// TwinCAT 3 PLC project Nonplanar_Master
// ProgramVersion: 3.1.4026.20
// libraries:
//   CmpBitmapPool, * (System)
//   Tc2_ControllerToolbox, * (Beckhoff Automation GmbH)
//   Tc2_DataExchange, * (Beckhoff Automation GmbH)
//   Tc2_SerialCom, * (Beckhoff Automation GmbH)
//   Tc2_Standard, * (Beckhoff Automation GmbH)
//   Tc2_System, * (Beckhoff Automation GmbH)
//   Tc2_Utilities, * (Beckhoff Automation GmbH)
//   VisuDialogs, * (System)
//   VisuSymbols,3.5.10.0,System
// project tree:
//   DUTs/ E_NozzleSizeFlow.TcDUT, E_StateExtruder.TcDUT, E_StateSequencer.TcTLEO, ST_ExtruderControl.TcDUT, ST_Hardware_IStepper.TcDUT, ST_HeaterZone.TcDUT, ST_HeaterZone_Parameter.TcDUT, ST_MaterialSettings.TcDUT, ST_MotorControl.TcDUT, ST_PrintingBed.TcDUT, ST_ProgramSequencer.TcDUT, ST_Hardware_QStepper.TcDUT
//   / GlobalTextList.TcGTLO, PlcTask.TcTTO, Visualisierungsmanager.TcVMO (not stored), VISU_TASK.TcTTO
//   GVLs/ GVL_ProgramSequencer.TcGVL, GVL_Instances.TcGVL
//   POUs/Extruder/ FB_ExtruderControl.TcPOU, FB_MotorControl.TcPOU, FB_HeaterZone.TcPOU, FC_ExtrusionCalculations.TcPOU, GVL_Extruder.TcGVL, GVL_HardwareExtruder.TcGVL, GVL_ParameterExtruder.TcGVL, PAR_Extruder.TcGVL
//   POUs/ FB_ProgramSequencer.TcPOU, FC_Instances.TcPOU, MAIN.TcPOU
//   POUs/HexaBridge/ FC_Execute.TcPOU, FC_ExecuteNoWait.TcPOU, FC_WaitForFinish.TcPOU, FC_WriteProgLine.TcPOU, GVL_HexaBridge.TcGVL
//   POUs/PrintingBed/ FB_PrintingBedSync.TcPOU, GVL_PrintingBed.TcGVL
//   VISUs/ ImagePool.TcIPO (not stored), V_Konfiguration.TcVIS, V_Homescreen.TcVIS
// real-time tasks:
//   TASK PlcTask: cycle T#10ms, priority 20, ADS port 350
//   TASK VISU_TASK: cycle T#200000us, priority 30, ADS port 351
// I/O:
//   DEVICE Gerät 1 (EtherCAT) (disabled), AmsNetId 172.16.4.140.2.1
//     Buskoppler Extruder (EK1100) [EK1100 EtherCAT-Koppler (2A E-Bus)]
//       Eingänge (EL1008) [EL1008 8K. Dig. Eingang 24V, 3ms]
//       Ausgänge SSR (EL2004) [EL2004 4K. Dig. Ausgang 24V, 0.5A]
//       Temperatursensoren (EL3204) [EL3204 4Ch. Ana. Input PT100 (RTD)]
//       Stepper Driver STEP (EL2521) [EL2521 1K. Pulse Train Ausgang]
//       Stepper Driver DIR / Enable (EL4132) [EL4132 2Ch. Ana. Ausgang +/-10V, 16bit]
//       Klemme 13 (EL9011) [EL9011 Endklemme]
// variable links:
//   Nonplanar_Master/Nonplanar_Master Instance <-> Device 1 (EtherCAT)/Buskoppler Extruder (EK1100)/Ausgänge SSR (EL2004)
//     PlcTask Outputs/GVL_HardwareExtruder.Q_Activate_Heaters <-> Channel 4/Output
//     PlcTask Outputs/GVL_HardwareExtruder.Q_SSR_Middle <-> Channel 2/Output
//     PlcTask Outputs/GVL_HardwareExtruder.Q_SSR_Nozzle <-> Channel 3/Output
//     PlcTask Outputs/GVL_HardwareExtruder.Q_SSR_Top <-> Channel 1/Output
//   Nonplanar_Master/Nonplanar_Master Instance <-> Device 1 (EtherCAT)/Buskoppler Extruder (EK1100)/Eingänge (EL1008)
//     PlcTask Inputs/GVL_HardwareExtruder.I_PelletsEmpty <-> Channel 1/Input
//   Nonplanar_Master/Nonplanar_Master Instance <-> Device 1 (EtherCAT)/Buskoppler Extruder (EK1100)/Stepper Driver DIR / Enable (EL4132)
//     PlcTask Outputs/GVL_HardwareExtruder.Q_Stepper/nDirection <-> Channel 1/Output
//     PlcTask Outputs/GVL_HardwareExtruder.Q_Stepper/nEnable <-> Channel 2/Output
//   Nonplanar_Master/Nonplanar_Master Instance <-> Device 1 (EtherCAT)/Buskoppler Extruder (EK1100)/Stepper Driver STEP (EL2521)
//     PlcTask Inputs/GVL_HardwareExtruder.I_Stepper/bError <-> PTO Status/Status/Error
//     PlcTask Inputs/GVL_HardwareExtruder.I_Stepper/bStallguardActive <-> PTO Status/Status/Status of input target
//     PlcTask Outputs/GVL_HardwareExtruder.Q_Stepper/nFrequencyValue <-> PTO Control/Frequency value
//   Nonplanar_Master/Nonplanar_Master Instance <-> Device 1 (EtherCAT)/Buskoppler Extruder (EK1100)/Temperatursensoren (EL3204)
//     PlcTask Inputs/GVL_HardwareExtruder.I_TempRaw_Middle <-> RTD Inputs Channel 2/Value
//     PlcTask Inputs/GVL_HardwareExtruder.I_TempRaw_Nozzle <-> RTD Inputs Channel 3/Value
//     PlcTask Inputs/GVL_HardwareExtruder.I_TempRaw_Top <-> RTD Inputs Channel 1/Value

CONFIGURATION Nonplanar_Master
    RESOURCE PLC ON TwinCAT3
        TASK PlcTask(INTERVAL := T#10ms, PRIORITY := 20);
        TASK VISU_TASK(INTERVAL := T#200000us, PRIORITY := 30);
        PROGRAM MAIN WITH PlcTask : MAIN;
        PROGRAM VisuElems_Visu_Prg WITH VISU_TASK : VisuElems.Visu_Prg;
    END_RESOURCE
END_CONFIGURATION

// ---- DUTs/E_NozzleSizeFlow.TcDUT
{attribute 'qualified_only'}
{attribute 'strict'}
// Düsendurchmesser in mm und die zugehärige Reduzierung des maximalen Durchflusses in mm^3/s
TYPE E_NozzleSizeFlow :
(
	fuenf 	:= 0,
	vier	:= -60,
	drei	:= -120,
	zwei 	:= -180,
	ein		:= -240
)DINT := drei;
END_TYPE

// ---- DUTs/E_StateExtruder.TcDUT
{attribute 'qualified_only'}
{attribute 'strict'}
TYPE E_StateExtruder :
(
	OFF			:= 0,
	INIT		:= 10,
	IDLE		:= 100,
	HEATING		:= 200,
	READY		:= 300,
	PRINTING	:= 310,
	SHUTDOWN	:= 400
);
END_TYPE

// ---- DUTs/E_StateSequencer.TcTLEO
{attribute 'qualified_only'}
{attribute 'strict'}
TYPE E_StateSequencer :
(
	OFF					:= 0,
	INIT_1				:= 10,
	INIT_2				:= 11,
	INIT_3				:= 12,
	HOMING_1			:= 90,
	HOMING_2			:= 91,
	
	IDLE				:= 100,
	OPEN_FILE			:= 110,
	CLOSE_FILE			:= 120,
	CHANGE_MATERIAL_1	:= 130,
	CHANGE_MATERIAL_2	:= 131,
	CHANGE_MATERIAL_3	:= 132,
	
	READY				:= 200,
	
	PREP_PRINTING		:= 300,
	PREP_PRINTING_HEX_1	:= 301,
	PREP_PRINTING_HEX_2	:= 302,
	PREP_PRINTING_HEX_3	:= 303,
	PREP_PRINTING_HEX_4 := 304,
	PREP_PRINTING_EXT	:= 305,
	PREP_PRINTING_HEX_5	:= 306,
	PREP_PRINTING_HEX_6	:= 307,
	PREP_PRINTING_HEX_7	:= 308,
	
	READ_FILE			:= 310,
	EXECUTE_LINE		:= 320,
	
	WRITE_KOS			:= 330,
	WRITE_FEED			:= 331,
	WRITE_PROG			:= 335,
	
	EXTRUDER_ON_1		:= 340,
	EXTRUDER_ON_2		:= 341,
	
	EXTRUDER_OFF_1		:= 350,
	START_EXTRUDING		:= 351,
	EXTRUDER_OFF_2		:= 352,
	
	STOP_EXTRUDING		:= 360,
	
	PAUSE				:= 390,
	
	ABORTED				:= 400,
	
	FINISHED			:= 500,
	
	SHUTDOWN			:= 600
);
END_TYPE

// ---- DUTs/ST_ExtruderControl.TcDUT
TYPE ST_ExtruderControl :
STRUCT
	// Steuersignale
	bErrorReset 	: BOOL;						// Reset-Befehl für Fehler
	bStartHeater 	: BOOL;						// Heizelemente aktivieren
	bStopHeater		: BOOL;						// Abschalten und Abkühlen
	bStart 			: BOOL;						// Start-Befehl Extrusion
	bStop 			: BOOL;						// Stop-Befehl Extrusion
	
	// Statusinformationen
	bReady 			: BOOL;						// Betriebsbereit
	bExtruding 		: BOOL;						// Motor läuft
	bHeatingActiv 	: BOOL;						// Heizelemente
	bError 			: BOOL;						// Fehler
	nErrorID      	: UDINT;
    sErrorMsg 		: STRING(80);
END_STRUCT
END_TYPE

// ---- DUTs/ST_Hardware_IStepper.TcDUT
TYPE ST_Hardware_IStepper :
STRUCT
	bStallguardActive 	: BOOL;		// Stallguard nicht aktive --> Motor überlastet
	bError				: BOOL;		// Fehler 
END_STRUCT
END_TYPE

// ---- DUTs/ST_HeaterZone.TcDUT
TYPE ST_HeaterZone :
STRUCT
    // Grunddaten
    bEnabled        : BOOL;                 // Zone aktiv
	fActualTemp   	: LREAL;             	// Isttemperatur [°C]
    fPID_Output     : LREAL;                // PID-Stellgröße [0..100%]
    bAtTemp         : BOOL;                 // Temperatur erreicht
	bErrorReset		: BOOL;					// Fehler zurücksetzen
    bError        	: BOOL;					// Fehler
    nErrorID      	: UDINT;
    sErrorMsg 		: STRING(80);
END_STRUCT
END_TYPE

// ---- DUTs/ST_HeaterZone_Parameter.TcDUT
TYPE ST_HeaterZone_Parameter :
STRUCT
    // PID-Parameter (https://docs.dyzedesign.com/pulsar.html#marlin-firmware)
    fKp             : LREAL 	:= 1.2;       	// Proportionalverstärkung
    fKi             : LREAL  	:= 0.015;   	// Integralverstärkung
    fKd             : LREAL  	:= 50.0;  		// Differentialversträrkung
    fFilterN      	: LREAL 	:= 10.0;		// Filterfaktor für DT1-Anteil des PID-Reglers (zwischen 5 und 20 --> mehr Rauschen = kleiner)
END_STRUCT
END_TYPE

// ---- DUTs/ST_MaterialSettings.TcDUT
TYPE ST_MaterialSettings :
STRUCT
	sMaterial		: STRING(80);		// Materialname	

	fTempPrintingBed: REAL	:= 0;		// <120 [°C]
	
	fTempTop		: LREAL	:= 0;		// <400 [°C]
	fTempMiddle		: LREAL	:= 0;		// <400 [°C]
	fTempNozzle		: LREAL	:= 0;		// <400 [°C]
	
	// https://docs.dyzedesign.com/pulsar.html#flow-to-rpm
	
	fMaxFlowRate	: LREAL := 0;		// Maximaler Volumenstrom [mm^3/s]
	fFlow2RPM		: LREAL := 0;		// Flow to RPM Ratio
	fNozzleSizeCoef	: LREAL := 1;		// Koeffizent Flow2RPM (abhängig von Material und Düse)
END_STRUCT	
END_TYPE

// ---- DUTs/ST_MotorControl.TcDUT
TYPE ST_MotorControl :
STRUCT
	bEnable         	: BOOL		:= FALSE;  	// Freigabe des Motors
	bErrorReset			: BOOL		:= FALSE;	// Fehler zurücksetzen
	bRunning       		: BOOL;					// Motor läuft
	bError        		: BOOL;					// Fehler
    nErrorID      		: UDINT;
    sErrorMsg 			: STRING(80);
END_STRUCT
END_TYPE

// ---- DUTs/ST_PrintingBed.TcDUT
TYPE ST_PrintingBed :
STRUCT
	fSetTemp		: REAL;			// Solltemperatur Druckbett
	fActualTemp		: REAL;			// Isttemperatur Druckbett
	bAtTemp			: BOOL;			// Solltemperatur erreicht (0.5°C Toleranz)
	bErrorReset		: BOOL;
	bError        	: BOOL;			// Fehler
    nErrorID      	: UDINT;
    sErrorMsg 		: STRING(80);
END_STRUCT
END_TYPE

// ---- DUTs/ST_ProgramSequencer.TcDUT
TYPE ST_ProgramSequencer :
STRUCT
	sPath			: STRING(MAX_STRING_LENGTH);// Pfad des Speicherorts des GeoCodes
	
	// Statusinformationen
	bReady 			: BOOL;						// Betriebsbereit
	bPrinting 		: BOOL;						// Druckprozess läuft
	bFinished		: BOOL;						// Druck abgeschlossen
	bError        	: BOOL;						// Fehler
    nErrorID      	: UDINT;
    sErrorMsg 		: STRING(80);
	
	// Steuersignale
	bHeatersEnabled	: BOOL;						// Heizelemente aktiviert --> später Safety Verknüpfung
	bPrintBedClear	: BOOL;						// Druckbett frei?
	bChangeMaterial	: BOOL;						// Extruder starten für Materialwechsel
	bChangeMaterialFinished : BOOL;				// Materialwechsel abschliesen und Extruder anhalten
	bLoadFile		: BOOL;						// File laden
	bCloseFile		: BOOL;						// File schließen
	bStart 			: BOOL;						// Start-Befehl
	bAbort 			: BOOL;						// Drucken abbrechen
	bPause          : BOOL;						// Pausiert Druckprozess
	bResume         : BOOL;						// Druckprozess fortsetzen
	bErrorReset 	: BOOL;						// Reset-Befehl für Fehler
END_STRUCT
END_TYPE

// ---- DUTs/ST_Hardware_QStepper.TcDUT
TYPE ST_Hardware_QStepper :
STRUCT
	nFrequencyValue		: INT;		// Frequenzwert (Bewegunggeschwindigkeit und Richtung) !muss INT sein, nicht UINT!
	nDirection			: INT;		// Legt Bewegungsrichtung fest (16383 entspricht 5V --> gegen den urzeigersinn --> Extrusion, alternativ 0)
	nEnable				: INT;		// Deaktivert Motor wenn aktiv (16383 entspricht 5V --> Motor aus, alternativ 0 entspricht 0V --> Motor an) 
END_STRUCT
END_TYPE

// ---- GVLs/GVL_ProgramSequencer.TcGVL
{attribute 'qualified_only'}
VAR_GLOBAL
	Sequencer		: ST_ProgramSequencer := (sPath := 'C:\Users\Gereon\Desktop\MotionInterface\testpaths\testpath.geo'); 
END_VAR

// ---- GVLs/GVL_Instances.TcGVL
VAR_GLOBAL
	// Befehlsverarbeitung
	Sequencer			: FB_ProgramSequencer;
	
	// Druckbett
	PrintingBed			: FB_PrintingBedSync;

	// Extruder
	ExtruderControl		: FB_ExtruderControl; 
	
	// Heizelemente
	HeaterTop			: FB_HeaterZone;
	HeaterMiddle		: FB_HeaterZone;
	HeaterNozzle		: FB_HeaterZone;
	
	//Motor
	ExtruderMotor		: FB_MotorControl;
END_VAR

// ---- POUs/Extruder/GVL_Extruder.TcGVL
{attribute 'qualified_only'}
VAR_GLOBAL
	Extruder		: ST_ExtruderControl;
	HeaterTop		: ST_HeaterZone;
	HeaterMiddle	: ST_HeaterZone;	
	HeaterNozzle	: ST_HeaterZone;
	ExtruderMotor	: ST_MotorControl;
END_VAR

// ---- POUs/Extruder/GVL_HardwareExtruder.TcGVL
{attribute 'qualified_only'}
VAR_GLOBAL
	// EL3204 – RTD-Temperatureingänge (Heizelemente)
	I_TempRaw_Top  		AT %I* : INT;  
	I_TempRaw_Middle 	AT %I* : INT;   
	I_TempRaw_Nozzle  	AT %I* : INT;    

	// EL2004 – Digitale Ausgänge (Heizelemente)
	Q_SSR_Top      		AT %Q* : BOOL;   
	Q_SSR_Middle    	AT %Q* : BOOL;   
	Q_SSR_Nozzle    	AT %Q* : BOOL;  
	Q_Activate_Heaters	AT %Q* : BOOL;

	// EL2521 – Pulsausgabe (Stepper Motor Driver)
	Q_Stepper	  		AT %Q* : ST_Hardware_QStepper;		
	I_Stepper  			AT %I* : ST_Hardware_IStepper;
	
	// EL1002 – Digitale Eingänge
	I_PelletsEmpty      AT %I* : BOOL;    	//Materialzuführung leer
END_VAR

// ---- POUs/Extruder/GVL_ParameterExtruder.TcGVL
{attribute 'qualified_only'}
VAR_GLOBAL PERSISTENT // Speichern der Online-Veränderungen
	// Mehr Informationen unter: https://docs.dyzedesign.com/pulsar.html#slicer-and-print-settings	

	// Materialabhängige Eigenschaften
	{attribute 'TcInitOnReset'} // Neuladen bei Kalt Reset (oben rechts)
	aMaterialSettings	: ARRAY[1..20] OF ST_MaterialSettings := [
			(sMaterial := 'Test-Material', 	fTempPrintingBed := 30, fTempTop := 201, 	fTempMiddle := 201, fTempNozzle := 201,	fMaxFlowRate := 600, fFlow2RPM := 0.65, fNozzleSizeCoef := 1.10),
			(sMaterial := 'PETG', 			fTempPrintingBed := 90, fTempTop := 101, 	fTempMiddle := 241, fTempNozzle := 231, fMaxFlowRate := 592, fFlow2RPM := 0.75,	fNozzleSizeCoef := 1.10),
			(sMaterial := 'PLA', 			fTempPrintingBed := 60, fTempTop := 101, 	fTempMiddle := 221, fTempNozzle := 211, fMaxFlowRate := 607, fFlow2RPM := 0.55,	fNozzleSizeCoef := 1.35),
			(sMaterial := 'PC-ABS-CF', 		fTempPrintingBed := 110,fTempTop := 301, 	fTempMiddle := 301, fTempNozzle := 301, fMaxFlowRate := 700, fFlow2RPM := 0.58, fNozzleSizeCoef := 1.10),
			(sMaterial := 'ABS', 			fTempPrintingBed := 90,	fTempTop := 131	, 	fTempMiddle := 231, fTempNozzle := 231, fMaxFlowRate := 658, fFlow2RPM := 0.65, fNozzleSizeCoef := 1.05), 
			15(())]; // Speichert materialabhängige Extrudereinstellungen (neues Material: Zeile oben kopieren, einfügen und Zähler reduzieren)		
	{attribute 'TcInitOnReset'} // Neuladen bei Kalt Reset (oben rechts)
	nMaterial		: UINT				:= 5;			// Aktuell gewähltes Material
		
	nNozzleSize		: E_NozzleSizeFlow	:= E_NozzleSizeFlow.vier; // Düsendurchmesser [mm] als Wort entspricht der Reduzierung des Durchflusses [mm^3/s]
	fLayerWidth     : LREAL 			:= 5.0;			// Schichtbreite [mm]
	fLayerHeight    : LREAL 			:= 1.0;			// Schichthöhe [mm]
	fSpeedOverride  : LREAL 			:= 10.0; 		// [%] Geschwindigkeits-Override in Prozent der Maximalgeschwindigkeit
	fSafetyMargin	: LREAL				:= 75.0;		// [%] Sicherheitsfaktor für die maximale Druckgeschwindigkeit (75%)
	
	// Berechnete Werte - siehe FC_ExtrusionCalculation
	fMaximumFlow	: LREAL				:= 0;			// Maximaler Durchfluss mit Abzug der Beschränkungen durch die Düse [mm^3/s]
	fMaximumSpeed	: LREAL				:= 0;			// Maximale Druckgeschwindigkeit [mm/s]
	fFlowRate		: LREAL				:= 0;			// Durchfluss [mm^3/s]
	fMotorRPM		: LREAL				:= 0;			// Notwendige RPM des Motors
	
	// Verfahrgeschwindigkeit
	fTravelSpeed	: LREAL				:= 100;			// Verfahrgeschwindigkeit [mm/s]
	
	// PID-Regler Heizelemente
	WarmupHeaterTop		: ST_HeaterZone_Parameter;
	WarmupHeaterMiddle	: ST_HeaterZone_Parameter;	
	WarmupHeaterNozzle	: ST_HeaterZone_Parameter;
	PrintingHeaterTop	: ST_HeaterZone_Parameter;
	PrintingHeaterMiddle: ST_HeaterZone_Parameter;	
	PrintingHeaterNozzle: ST_HeaterZone_Parameter;
	
	tRampTime		: TIME				:= T#3M;		// Länge der Rampe bei Sprüngen
	nPIDCycleFactor	: UINT  			:= 10;			// PID rechnet alle n Zyklen
    tPWM_Period     : TIME  			:= T#3S;        // PWM-Periode SSR
    fAtTempTolerance: LREAL 			:= 50.0;         // Toleranz für Signal Temperatur erreicht [°C]
END_VAR

// ---- POUs/Extruder/PAR_Extruder.TcGVL
{attribute 'qualified_only'}
VAR_GLOBAL CONSTANT
	// Nicht bearbeiten!
	// Quelle: https://docs.dyzedesign.com/pulsar.html#marlin-firmware	

	// Temperatur
    C_MAX_SET_TEMP		: LREAL := 400.0;		// Maximale Setzbare Temperaturgrenze [°C]
    C_MIN_SET_TEMP		: LREAL := 0;			// Minimal Setzbare Temperaturgrenze [°C]
	C_MAX_SENSOR_TEMP	: LREAL := 505.0;		// Maximale Plausibilitätsgrenze Sensoren [°C]
    C_MIN_SENSOR_TEMP	: LREAL := 0;			// Minimale Plausibilitätsgrenze Sensoren [°C]
	C_MAX_TEMP			: LREAL := 500.0;		// Maximaltemperatur Extruder [°C]
	
	// Stepper Driver 
	C_MAX_RPM_SCREW		: LREAL := 60;			// Maximale zulässige RPM --> Anpassung: EL2521 Grundfrequenz
	C_MAX_RPM_SCREW_FULL: LREAL := 50;			// Maximale zulässige RPM mit Material
	C_GEAR_RATIO		: LREAL := 11.46;		// Übersetzung Motor --> Schraube
	C_STEPPER_DIR		: BOOL	:= FALSE;		// Drehrichtung
END_VAR

// ---- POUs/HexaBridge/GVL_HexaBridge.TcGVL
{attribute 'qualified_only' := 'FALSE'}
//  GVL_HexaBridge  -  Globale Variablen für ADS-HexaBOF-Bridge
VAR_GLOBAL
    // Befehlsschnittstelle
    sCommand        : STRING(255);          // Befehlsname
    sParameter      : STRING(1000);         // Parameter-String
    bExecute        : BOOL;                 // Steigende Flanke = Befehl ausführen
	bCommandSent	: BOOL;					// Befehl gesendet
    bBusy           : BOOL;                 // Bridge verarbeitet Befehl
    bDone           : BOOL;                 // Befehl abgeschlossen
    bError          : BOOL;                 // Fehler aufgetreten
    nErrorCode      : INT;                  // Fehlercode (0=OK)
    sErrorMsg       : STRING(255);          // Fehlermeldung
    sResult         : STRING(1000);         // Ergebnis-String

    // Status
    bHexConnected   : BOOL;                 // HexaBOF verbunden
    bBridgeRunning  : BOOL;                 // Python-Bridge aktiv

    // Direkte GEO-Strings
    sGeoLine        : STRING(1000);         // Einzel-GEO-Zeile
    sGeoBlock       : STRING(10000);        // GEO-Block (mehrzeilig)
	
	// Programm Block schreiben im Hintergrund, um diesen später auszuführen
	sProgLine		: STRING(1000);         // Einzel-GEO-Zeile zu Programm hinzufügen
	bProgLineReady	: BOOL;        			// Zeile bereit zum schreiben
	bProgLineSaved	: BOOL;        			// Zeile gespeichert
	bProgLineExecution : BOOL;        		// Blockiert das Schreiben neuer Programmzeilen beim Starten des Ausführens eines Blocks
END_VAR

// ---- POUs/PrintingBed/GVL_PrintingBed.TcGVL
{attribute 'qualified_only'}
VAR_GLOBAL
	PrintingBed		: ST_PrintingBed;
END_VAR

// ---- POUs/MAIN.TcPOU
PROGRAM MAIN
VAR
END_VAR

FC_Instances();

END_PROGRAM

// ---- POUs/FC_Instances.TcPOU
FUNCTION FC_Instances : BOOL
VAR_INPUT
END_VAR
VAR
END_VAR

// Befehlsverarbeitung
Sequencer(
	sPath			:= GVL_ProgramSequencer.Sequencer.sPath,
	bPelletsEmpty	:= GVL_HardwareExtruder.I_PelletsEmpty,
	bReady 			=> GVL_ProgramSequencer.Sequencer.bReady,
	bPrinting 		=> GVL_ProgramSequencer.Sequencer.bPrinting,
	bFinished		=> GVL_ProgramSequencer.Sequencer.bFinished,
	bError        	=> GVL_ProgramSequencer.Sequencer.bError,
	nErrorID      	=> GVL_ProgramSequencer.Sequencer.nErrorID,
	sErrorMsg 		=> GVL_ProgramSequencer.Sequencer.sErrorMsg,
	bHeatersEnabled	:= GVL_ProgramSequencer.Sequencer.bHeatersEnabled,
	bPrintBedClear	:= GVL_ProgramSequencer.Sequencer.bPrintBedClear,
	bChangeMaterial	:= GVL_ProgramSequencer.Sequencer.bChangeMaterial,
	bChangeMaterialFinished := GVL_ProgramSequencer.Sequencer.bChangeMaterialFinished,
	bLoadFile		:= GVL_ProgramSequencer.Sequencer.bLoadFile,
	bCloseFile		:= GVL_ProgramSequencer.Sequencer.bCloseFile,
	bStart 			:= GVL_ProgramSequencer.Sequencer.bStart,
	bAbort 			:= GVL_ProgramSequencer.Sequencer.bAbort,
	bPause          := GVL_ProgramSequencer.Sequencer.bPause,
	bResume         := GVL_ProgramSequencer.Sequencer.bResume,
	bErrorReset 	:= GVL_ProgramSequencer.Sequencer.bErrorReset);

// Druckbett
PrintingBed(
	bErrorReset		:= GVL_PrintingBed.PrintingBed.bErrorReset,
	bError			=> GVL_PrintingBed.PrintingBed.bError,
	nErrorID		=> GVL_PrintingBed.PrintingBed.nErrorID,
	sErrorMsg		=> GVL_PrintingBed.PrintingBed.sErrorMsg);

// Extruder	
ExtruderControl(
	bErrorReset		:= GVL_Extruder.Extruder.bErrorReset,
	bHeatersEnabled := GVL_ProgramSequencer.Sequencer.bHeatersEnabled,
	bReady			=> GVL_Extruder.Extruder.bReady,
	bExtruding		=> GVL_Extruder.Extruder.bExtruding,
	bHeatingActiv	=> GVL_Extruder.Extruder.bHeatingActiv,
	bError			=> GVL_Extruder.Extruder.bError,
	nErrorID      	=> GVL_Extruder.Extruder.nErrorID,
    sErrorMsg 		=> GVL_Extruder.Extruder.sErrorMsg,
	bStartHeater	:= GVL_Extruder.Extruder.bStartHeater,
	bStopHeater		:= GVL_Extruder.Extruder.bStopHeater,
	bStart			:= GVL_Extruder.Extruder.bStart,
	bStop			:= GVL_Extruder.Extruder.bStop);	

// Heizelemente
HeaterTop(
	bEnable			:= GVL_Extruder.HeaterTop.bEnabled,
    fSetTemp		:= GVL_ParameterExtruder.aMaterialSettings[GVL_ParameterExtruder.nMaterial].fTempTop,
	fPID_Output     => GVL_Extruder.HeaterTop.fPID_Output,
	bAtTemp         => GVL_Extruder.HeaterTop.bAtTemp,
    bErrorReset		:= GVL_Extruder.HeaterTop.bErrorReset,
    bError        	=> GVL_Extruder.HeaterTop.bError,
    nErrorID      	=> GVL_Extruder.HeaterTop.nErrorID,
    sErrorMsg 		=> GVL_Extruder.HeaterTop.sErrorMsg,
	fWarmupKp       := GVL_ParameterExtruder.WarmupHeaterTop.fKp,
	fWarmupKi       := GVL_ParameterExtruder.WarmupHeaterTop.fKi,
	fWarmupKd       := GVL_ParameterExtruder.WarmupHeaterTop.fKd,
	fWarmupFilterN 	:= GVL_ParameterExtruder.WarmupHeaterTop.fFilterN,
	bPrinting		:= GVL_Extruder.Extruder.bExtruding,
	fPrintingKp     := GVL_ParameterExtruder.PrintingHeaterTop.fKp,
	fPrintingKi     := GVL_ParameterExtruder.PrintingHeaterTop.fKi,
	fPrintingKd     := GVL_ParameterExtruder.PrintingHeaterTop.fKd,
	fPrintingFilterN:= GVL_ParameterExtruder.PrintingHeaterTop.fFilterN,
	tRampTime		:= GVL_ParameterExtruder.tRampTime,
	nPIDCycleFactor	:= GVL_ParameterExtruder.nPIDCycleFactor,
	tPWM_Period     := GVL_ParameterExtruder.tPWM_Period,
	fAtTempTolerance:= GVL_ParameterExtruder.fAtTempTolerance,
	nTempRaw		:= GVL_HardwareExtruder.I_TempRaw_Top,
	fActualTemp		=> GVL_Extruder.HeaterTop.fActualTemp,
	bSSR_Out		=> GVL_HardwareExtruder.Q_SSR_Top);

HeaterMiddle(
	bEnable			:= GVL_Extruder.HeaterMiddle.bEnabled,
    fSetTemp		:= GVL_ParameterExtruder.aMaterialSettings[GVL_ParameterExtruder.nMaterial].fTempMiddle,
	fPID_Output     => GVL_Extruder.HeaterMiddle.fPID_Output,
	bAtTemp         => GVL_Extruder.HeaterMiddle.bAtTemp,
    bErrorReset		:= GVL_Extruder.HeaterMiddle.bErrorReset,
    bError        	=> GVL_Extruder.HeaterMiddle.bError,
    nErrorID      	=> GVL_Extruder.HeaterMiddle.nErrorID,
    sErrorMsg 		=> GVL_Extruder.HeaterMiddle.sErrorMsg,
	fWarmupKp       := GVL_ParameterExtruder.WarmupHeaterMiddle.fKp,
	fWarmupKi       := GVL_ParameterExtruder.WarmupHeaterMiddle.fKi,
	fWarmupKd       := GVL_ParameterExtruder.WarmupHeaterMiddle.fKd,
	fWarmupFilterN 	:= GVL_ParameterExtruder.WarmupHeaterMiddle.fFilterN,
	bPrinting		:= GVL_Extruder.Extruder.bExtruding,
	fPrintingKp     := GVL_ParameterExtruder.PrintingHeaterMiddle.fKp,
	fPrintingKi     := GVL_ParameterExtruder.PrintingHeaterMiddle.fKi,
	fPrintingKd     := GVL_ParameterExtruder.PrintingHeaterMiddle.fKd,
	fPrintingFilterN:= GVL_ParameterExtruder.PrintingHeaterMiddle.fFilterN,
	tRampTime		:= GVL_ParameterExtruder.tRampTime,
	nPIDCycleFactor	:= GVL_ParameterExtruder.nPIDCycleFactor,  
	tPWM_Period     := GVL_ParameterExtruder.tPWM_Period,      
	fAtTempTolerance:= GVL_ParameterExtruder.fAtTempTolerance,
	nTempRaw		:= GVL_HardwareExtruder.I_TempRaw_Middle,
	fActualTemp		=> GVL_Extruder.HeaterMiddle.fActualTemp,
	bSSR_Out		=> GVL_HardwareExtruder.Q_SSR_Middle);
		
HeaterNozzle(
	bEnable			:= GVL_Extruder.HeaterNozzle.bEnabled,
    fSetTemp		:= GVL_ParameterExtruder.aMaterialSettings[GVL_ParameterExtruder.nMaterial].fTempNozzle,
	fPID_Output     => GVL_Extruder.HeaterNozzle.fPID_Output,
	bAtTemp         => GVL_Extruder.HeaterNozzle.bAtTemp,
    bErrorReset		:= GVL_Extruder.HeaterNozzle.bErrorReset,
    bError        	=> GVL_Extruder.HeaterNozzle.bError,
    nErrorID      	=> GVL_Extruder.HeaterNozzle.nErrorID,
    sErrorMsg 		=> GVL_Extruder.HeaterNozzle.sErrorMsg,
	fWarmupKp       := GVL_ParameterExtruder.WarmupHeaterNozzle.fKp,
	fWarmupKi       := GVL_ParameterExtruder.WarmupHeaterNozzle.fKi,
	fWarmupKd       := GVL_ParameterExtruder.WarmupHeaterNozzle.fKd,
	fWarmupFilterN 	:= GVL_ParameterExtruder.WarmupHeaterNozzle.fFilterN,
	bPrinting		:= GVL_Extruder.Extruder.bExtruding,
	fPrintingKp     := GVL_ParameterExtruder.PrintingHeaterNozzle.fKp,
	fPrintingKi     := GVL_ParameterExtruder.PrintingHeaterNozzle.fKi,
	fPrintingKd     := GVL_ParameterExtruder.PrintingHeaterNozzle.fKd,
	fPrintingFilterN:= GVL_ParameterExtruder.PrintingHeaterNozzle.fFilterN,
	tRampTime		:= GVL_ParameterExtruder.tRampTime,
	nPIDCycleFactor	:= GVL_ParameterExtruder.nPIDCycleFactor,  
	tPWM_Period     := GVL_ParameterExtruder.tPWM_Period,      
	fAtTempTolerance:= GVL_ParameterExtruder.fAtTempTolerance,
	nTempRaw		:= GVL_HardwareExtruder.I_TempRaw_Nozzle,
	fActualTemp		=> GVL_Extruder.HeaterNozzle.fActualTemp,
	bSSR_Out		=> GVL_HardwareExtruder.Q_SSR_Nozzle);

//Motor
ExtruderMotor(
	bEnable			:= GVL_Extruder.ExtruderMotor.bEnable,
	bErrorReset		:= GVL_Extruder.ExtruderMotor.bErrorReset,
	fSetRPM			:= GVL_ParameterExtruder.fMotorRPM,
	bError_Stepper	:= GVL_HardwareExtruder.I_Stepper.bError,
	bStepper_STALL	:= GVL_HardwareExtruder.I_Stepper.bStallguardActive,
	bRunning		=> GVL_Extruder.ExtruderMotor.bRunning,
	bError			=> GVL_Extruder.ExtruderMotor.bError,
	nErrorID		=> GVL_Extruder.ExtruderMotor.nErrorID,
	sErrorMsg		=> GVL_Extruder.ExtruderMotor.sErrorMsg,
	nPTO_FreqValue	=> GVL_HardwareExtruder.Q_Stepper.nFrequencyValue,
	n_Direction		=> GVL_HardwareExtruder.Q_Stepper.nDirection,
	n_Enable		=> GVL_HardwareExtruder.Q_Stepper.nEnable);

END_FUNCTION

// ---- POUs/FB_ProgramSequencer.TcPOU
FUNCTION_BLOCK FB_ProgramSequencer
VAR_INPUT
	sPath			: STRING(MAX_STRING_LENGTH);// Pfad des Speicherorts des GeoCodes
	bPelletsEmpty	: BOOL;						// Feeding System meldet, dass keine Pellets am Extruder ankommen
END_VAR
VAR_OUTPUT
	// Statusinformationen
	bReady 			: BOOL;						// Betriebsbereit
	bPrinting 		: BOOL;						// Druckprozess läuft
	bFinished		: BOOL;						// Druck abgeschlossen
	bError        	: BOOL;						// Fehler
    nErrorID      	: UDINT;
    sErrorMsg 		: STRING(80);
END_VAR
VAR
	// Zustandsmaschine
	eState			: E_StateSequencer := E_StateSequencer.OFF;	// Zustand
	eLastState		: E_StateSequencer := E_StateSequencer.OFF; // Vorheriger zustand
	bFirstRunState	: BOOL;						// Erster Durchlauf des Zusands nach einem Zusandswechsel
	
	// Dateiverarbeitung
	fbOpenFile		: FB_FileOpen;
	fbReadFile		: FB_FileGets;
	fbCloseFile		: FB_FileClose;
	hFile  			: UINT;						// file handle
	bFileLoaded		: BOOL;						// Datei geladen
	sLine 			: STRING(MAX_STRING_LENGTH);// Speicher für die gelesene Zeile
	sLineTrimmed	: STRING(MAX_STRING_LENGTH);
	
	// Programmablauf
	bProgBlockStart			: BOOL;				// Erster Befehl des Programmblocks
	bBlockWithExt			: BOOL;				// Extruder in Programmblock aktiv
	bStopExtOnBlockEnd 		: BOOL;				// Extruder am Blockende ausschalten
	bBackToExtruderOn2	 	: BOOL;				// Rücksprung nach Anhalten des Extruders
	bBackToPause			: BOOL;				// Rücksprung nach Anhalten des Extruders
	
	// Änderung Vorschubgeschwindigkeit
	fFeed			: LREAL;
	fTravelFeed		: LREAL;
	bDryRun: BOOL := TRUE;
END_VAR
VAR_IN_OUT
	// Steuersignale
	bHeatersEnabled	: BOOL;						// Heizelemente aktiviert
	bPrintBedClear	: BOOL;						// Druckbett frei?
	bChangeMaterial	: BOOL;						// Extruder starten für Materialwechsel
	bChangeMaterialFinished : BOOL;				// Materialwechsel abschliesen und Extruder anhalten
	bLoadFile		: BOOL;						// File laden
	bCloseFile		: BOOL;						// File schließen
	bStart 			: BOOL;						// Start-Befehl
	bAbort 			: BOOL;						// Drucken abbrechen
	bPause          : BOOL;						// Pausiert Druckprozess
	bResume         : BOOL;						// Druckprozess fortsetzen
	bErrorReset 	: BOOL;						// Reset-Befehl für Fehler
END_VAR

// Schritte: DUTs/E_StateSequencer

// =============================================================================
// Zustandsmaschine
// =============================================================================
IF eLastState <> eState THEN
	bFirstRunState := TRUE;
ELSE
	bFirstRunState := FALSE;
END_IF
eLastState := eState;

// =============================================================================
// Funktionsabhängigkeiten
// =============================================================================
IF bPelletsEmpty THEN
	bPause := TRUE;
	sErrorMsg := 'Feeding System meldet, dass keine Pellets am Extruder ankommen';
END_IF

IF bAbort OR bPause THEN
	bStart := FALSE;
END_IF

IF NOT bHeatersEnabled THEN
	GVL_Extruder.Extruder.bStopHeater := TRUE;
END_IF

IF bResume THEN
	bPause := FALSE;
END_IF

GVL_HardwareExtruder.Q_Activate_Heaters := bHeatersEnabled;

// =============================================================================
// Fehlerbahandlung
// =============================================================================

// Da absolut nichts angeschlossen ist, zwingen wir im Trockenlauf ALLE 
// Hardware-Komponenten auf "fehlerfrei" und "betriebsbereit"!
IF bDryRun THEN
	
	// A. HexaBridge Spoofing
	GVL_HexaBridge.bError := FALSE;
	GVL_HexaBridge.nErrorCode := 0;
	GVL_HexaBridge.sErrorMsg := '';
	GVL_HexaBridge.bHexConnected := TRUE;
	GVL_HexaBridge.bBridgeRunning := TRUE;
	
	// B. Extruder Spoofing (Fehlerfrei & sofort heiß)
	GVL_Extruder.Extruder.bError := FALSE;
	GVL_Extruder.Extruder.nErrorID := 0;
	GVL_Extruder.Extruder.sErrorMsg := '';
	GVL_Extruder.Extruder.bReady := TRUE;
	// Wenn TwinCAT heizen will, tun wir so, als wäre er sofort heiß:
	IF bHeatersEnabled THEN 
		GVL_Extruder.Extruder.bHeatingActiv := TRUE; 
	END_IF

	// C. Druckbett Spoofing (Fehlerfrei & Zieltemperatur erreicht)
	GVL_PrintingBed.PrintingBed.bError := FALSE;
	GVL_PrintingBed.PrintingBed.nErrorID := 0;
	GVL_PrintingBed.PrintingBed.sErrorMsg := '';
	// Wenn eine Zieltemperatur > 0 gesetzt wird, geben wir sofort das "Ist warm!" Signal:
	IF GVL_PrintingBed.PrintingBed.fSetTemp > 0.0 THEN
		GVL_PrintingBed.PrintingBed.bAtTemp := TRUE;
	ELSE
		GVL_PrintingBed.PrintingBed.bAtTemp := FALSE;
	END_IF

END_IF


// Fehler zurücksetzen
IF bErrorReset AND bError THEN
	GVL_Extruder.Extruder.bErrorReset := TRUE;
	GVL_PrintingBed.PrintingBed.bErrorReset := TRUE;
	
	// HexaBridge reset
	GVL_HexaBridge.bExecute := FALSE;
	GVL_HexaBridge.bError := FALSE;
	GVL_HexaBridge.nErrorCode := 0;
	GVL_HexaBridge.sErrorMsg := '';
	
	bErrorReset := FALSE;
	bError := FALSE;
	nErrorID := 0;
	sErrorMsg := '';
ELSIF bErrorReset AND NOT bError THEN
	sErrorMsg := '';
END_IF

// Fehler zusammenführen
bError := bError 
	OR GVL_Extruder.Extruder.bError
	OR GVL_HexaBridge.bError
	OR GVL_PrintingBed.PrintingBed.bError;

// Fehlernachrichten zusammenführen
IF bError THEN
	IF GVL_Extruder.Extruder.bError			THEN nErrorID := GVL_Extruder.Extruder.nErrorID; END_IF
	IF GVL_HexaBridge.bError				THEN nErrorID := TO_UDINT(GVL_Hexabridge.nErrorCode); END_IF
	IF GVL_PrintingBed.PrintingBed.bError	THEN nErrorID := GVL_PrintingBed.PrintingBed.nErrorID; END_IF
	
	IF GVL_Extruder.Extruder.bError			THEN sErrorMsg := GVL_Extruder.Extruder.sErrorMsg; END_IF
	IF GVL_HexaBridge.bError				THEN sErrorMsg := GVL_Hexabridge.sErrorMsg; END_IF
	IF GVL_PrintingBed.PrintingBed.bError	THEN sErrorMsg := GVL_PrintingBed.PrintingBed.sErrorMsg; END_IF
END_IF

// Zusandswechsel im Fehlerfall
IF bError AND NOT (eState = E_StateSequencer.IDLE 
				OR eState = E_StateSequencer.OFF 
				OR eState = E_StateSequencer.READY
				OR eState = E_StateSequencer.SHUTDOWN) THEN
	IF eState < E_StateSequencer.IDLE THEN
		eState := E_StateSequencer.OFF;
	ELSIF eState > E_StateSequencer.READY AND eState < E_StateSequencer.ABORTED THEN
		GVL_Extruder.Extruder.bStopHeater := TRUE;
		bHeatersEnabled := FALSE;
		bAbort := TRUE;
		eState := E_StateSequencer.ABORTED;
	END_IF
END_IF

IF (NOT GVL_Hexabridge.bBridgeRunning OR NOT GVL_Hexabridge.bHexConnected)
AND eState >= E_StateSequencer.READY THEN
	eState := E_StateSequencer.OFF;
	bError := TRUE;
	sErrorMsg := 'HexaBridge ist nicht verbunden!';
END_IF

// =============================================================================
// Status
// =============================================================================
bPrinting := GVL_Extruder.Extruder.bExtruding OR GVL_Extruder.Extruder.bReady;

// =============================================================================
// Vorschubgeschwindigkeit
// =============================================================================
fFeed := GVL_ParameterExtruder.fMaximumSpeed;
fTravelFeed := GVL_ParameterExtruder.fTravelSpeed;

// =============================================================================
// Zustandsmaschine
// =============================================================================
CASE eState OF
	// =============================================================================
	E_StateSequencer.OFF : // Ausgeschaltet
	// =============================================================================
		// Alles aus
		GVL_Extruder.Extruder.bStartHeater := FALSE;
		GVL_Extruder.Extruder.bStopHeater := TRUE;
		GVL_Extruder.Extruder.bStart := FALSE;
		GVL_Extruder.Extruder.bStop := TRUE;
		GVL_PrintingBed.PrintingBed.fSetTemp := 0.0;
	
		// Status
		bReady := FALSE;
		
		IF NOT bError THEN
			eState := E_StateSequencer.INIT_1;
		END_IF
	
	// =============================================================================
	E_StateSequencer.INIT_1: // Initialisierung
	// =============================================================================
		IF GVL_HexaBridge.bHexConnected AND GVL_HexaBridge.bBridgeRunning THEN
			eState := E_StateSequencer.INIT_2;
		END_IF
		
	// =============================================================================
	E_StateSequencer.INIT_2: // Koordinatensystem setzen
	// =============================================================================
		IF FC_Execute('GEO_LINE','SK Extruder') THEN
			eState := E_StateSequencer.INIT_3;
		END_IF
		
	// =============================================================================
	E_StateSequencer.INIT_3: // Kardanwinkel auswählen
	// =============================================================================
		IF FC_Execute('GEO_LINE','NF 2') THEN
			eState := E_StateSequencer.HOMING_1;
		END_IF
	
	// =============================================================================
	E_StateSequencer.HOMING_1: // Verfahrgeschwindigkeit setzen
	// =============================================================================
		IF FC_Execute('GEO_LINE',CONCAT('VF ',TO_STRING(fTravelFeed * 60))) THEN // Vorschub [mm/min]
			eState := E_StateSequencer.HOMING_2;
		END_IF
	
	// =============================================================================
	E_StateSequencer.HOMING_2: // Home Position anfahren (Einfahren)
	// =============================================================================
		IF FC_Execute('GEO_LINE','PU') THEN
			eState := E_StateSequencer.IDLE;
		END_IF
	
	// =============================================================================
	E_StateSequencer.IDLE : // Idle (Keine Datei geöffnet)
	// =============================================================================
		// Alles aus
		GVL_Extruder.Extruder.bStartHeater := FALSE;
		GVL_Extruder.Extruder.bStart := FALSE;
	
		// Status
		bReady := FALSE;
		
		IF bChangeMaterial THEN
			eState := E_StateSequencer.CHANGE_MATERIAL_1;
		ELSIF bFileLoaded THEN 
			eState := E_StateSequencer.READY;
		ELSIF bLoadFile THEN
			eState := E_StateSequencer.OPEN_FILE;
		END_IF
	
	// =============================================================================
	E_StateSequencer.OPEN_FILE : // File öffnen
	// =============================================================================
		IF bFirstRunState THEN
			fbOpenFile(
				sNetId := '', 
				sPathName := sPath, 
				nMode := FOPEN_MODEREAD, 
				bExecute := TRUE, 
				tTimeout := T#5S);
		ELSE
			fbOpenFile(bExecute := FALSE);
		END_IF
			
		IF fbOpenFile.bError THEN
			bError := TRUE;
			nErrorID := 3001;
			sErrorMsg := 'Datei: Fehler beim oeffnen der Datei';
		END_IF
		
		IF NOT bFirstRunState AND NOT fbOpenFile.bBusy AND NOT fbOpenFile.bError AND fbOpenFile.hFile <> 0 THEN
			hFile := fbOpenFile.hFile;
			bFileLoaded := TRUE;
			bLoadFile := FALSE;
			eState := E_StateSequencer.READY;
		END_IF

	// =============================================================================
	E_StateSequencer.CLOSE_FILE : // File schließen
	// =============================================================================
		IF bFirstRunState AND hFile <> 0 THEN
			fbCloseFile(
				sNetId := '',
  				hFile := hFile,
				bExecute := TRUE, 
				tTimeout := T#5S);
		ELSE
			fbCloseFile(bExecute := FALSE);
		END_IF
		
		IF fbCloseFile.bError THEN
			bError := TRUE;
			nErrorID := 3002;
			sErrorMsg := 'Datei: Fehler beim schliessen der Datei';
		END_IF
		
		IF (NOT bFirstRunState AND NOT fbCloseFile.bBusy AND NOT fbCloseFile.bError) 
		OR hFile = 0 THEN
			hFile := 0;
			bFileLoaded := FALSE;
			bCloseFile := FALSE;
			eState := E_StateSequencer.IDLE;
		END_IF
		
	// =============================================================================
	E_StateSequencer.CHANGE_MATERIAL_1 : // Extruder aufheizen
	// =============================================================================
		bChangeMaterial := FALSE;
	
		// Heizungen aktivieren
		IF bHeatersEnabled THEN
			GVL_Extruder.Extruder.bStopHeater := FALSE;
			GVL_Extruder.Extruder.bStartHeater := TRUE;
		END_IF
		
		//Status
		bPrintBedClear := FALSE;
		
		IF bAbort THEN
			eState := E_StateSequencer.ABORTED;		
		ELSIF GVL_Extruder.Extruder.bReady THEN
			eState := E_StateSequencer.CHANGE_MATERIAL_2;
		END_IF
		
	// =============================================================================
	E_StateSequencer.CHANGE_MATERIAL_2 : // Extrudieren bis zum Beenden
	// =============================================================================
		// Extruder aktivieren
		GVL_Extruder.Extruder.bStop := FALSE;
		GVL_Extruder.Extruder.bStart := TRUE;
		bPrintBedClear := FALSE;
		
		IF bAbort THEN
			eState := E_StateSequencer.ABORTED;
		ELSIF bChangeMaterialFinished THEN
			bChangeMaterialFinished := FALSE;
			eState := E_StateSequencer.CHANGE_MATERIAL_3;
		END_IF
		
	// =============================================================================
	E_StateSequencer.CHANGE_MATERIAL_3 : // Extruder abschalten
	// =============================================================================
		GVL_Extruder.Extruder.bStop := TRUE;
		GVL_Extruder.Extruder.bStopHeater := TRUE;
		GVL_Extruder.Extruder.bStart := FALSE;
		GVL_Extruder.Extruder.bStartHeater := FALSE;
		IF NOT GVL_Extruder.Extruder.bExtruding THEN
			eState := E_StateSequencer.IDLE;
		END_IF
		
	// =============================================================================
	E_StateSequencer.READY: // Druckbereit, Programm geöffnet
	// =============================================================================
		//Status
		bReady := TRUE;
		bFinished := FALSE;
		
		IF NOT bFileLoaded THEN
			eState := E_StateSequencer.IDLE;
		ELSIF bCloseFile AND bFileLoaded THEN
			eState := E_StateSequencer.CLOSE_FILE;
		ELSIF bStart AND bPrintBedClear AND bHeatersEnabled
		AND GVL_Hexabridge.bBridgeRunning AND GVL_Hexabridge.bHexConnected THEN
			bStart := FALSE;
			eState := E_StateSequencer.PREP_PRINTING;
		END_IF
	
	// =============================================================================
	E_StateSequencer.PREP_PRINTING : // Werte zurücksetzen
	// =============================================================================
		bProgBlockStart := TRUE;
		bBlockWithExt := FALSE;
		bStopExtOnBlockEnd := FALSE;
		bBackToExtruderOn2 := FALSE;
		bBackToPause := FALSE;
		
		eState := E_StateSequencer.PREP_PRINTING_HEX_1;
		
	// =============================================================================
	E_StateSequencer.PREP_PRINTING_HEX_1: // Koordinatensystem setzen
	// =============================================================================
		IF FC_Execute('GEO_LINE','SK Extruder') THEN
			eState := E_StateSequencer.PREP_PRINTING_HEX_2;
		END_IF
		
	// =============================================================================
	E_StateSequencer.PREP_PRINTING_HEX_2 : // Druckprozess gestartet (Hexapod Geschwindigkeit setzen)
	// =============================================================================
		IF FC_Execute('GEO_LINE',CONCAT('VF ',TO_STRING(fTravelFeed * 60))) THEN // Verfahrgeschwindigkeit [mm/min]
			IF bAbort THEN
				eState := E_StateSequencer.ABORTED;
			ELSE
				eState := E_StateSequencer.PREP_PRINTING_HEX_3;
			END_IF
		END_IF
	
	// =============================================================================
	E_StateSequencer.PREP_PRINTING_HEX_3 : // Override überschreiben, um Fehler zu verhindern
	// =============================================================================
		IF FC_Execute('GEO_LINE','OV 1.0') THEN
			IF bAbort THEN
				eState := E_StateSequencer.ABORTED;
			ELSE
				eState := E_StateSequencer.PREP_PRINTING_HEX_4;
			END_IF
		END_IF		

	// =============================================================================
	E_StateSequencer.PREP_PRINTING_HEX_4 : // Druckprozess gestartet (Hexapod auf Eckposition fahren)
	// =============================================================================
		IF FC_Execute('GEO_LINE','LA 230 60 -200 0 0 0') THEN // Eckposition vorn
			IF bAbort THEN
				eState := E_StateSequencer.ABORTED;
			ELSE
				eState := E_StateSequencer.PREP_PRINTING_HEX_5;
			END_IF
		END_IF
	
	// =============================================================================
	E_StateSequencer.PREP_PRINTING_HEX_5 : // Druckprozess gestartet (Genauhalt deaktivieren, für flüssige Bewegungen)
	// =============================================================================
		IF FC_Execute('GEO_LINE','GH 0') THEN
			IF bAbort THEN
				eState := E_StateSequencer.ABORTED;
			ELSE
				eState := E_StateSequencer.PREP_PRINTING_EXT;
			END_IF
		END_IF
		
	// =============================================================================
	E_StateSequencer.PREP_PRINTING_EXT : // Druckprozess gestartet (Extruder und Druckbett aufheizen)
	// =============================================================================
		// Heizungen aktivieren
		IF bHeatersEnabled THEN
			GVL_PrintingBed.PrintingBed.fSetTemp := GVL_ParameterExtruder.aMaterialSettings[GVL_ParameterExtruder.nMaterial].fTempPrintingBed;
			GVL_Extruder.Extruder.bStopHeater := FALSE;
			GVL_Extruder.Extruder.bStartHeater := TRUE;
		END_IF
		
		//Status
		bReady := FALSE;
		bPrintBedClear := FALSE;
		
		IF bAbort THEN
			eState := E_StateSequencer.ABORTED;		
		ELSIF GVL_Extruder.Extruder.bReady AND GVL_Extruder.Extruder.bHeatingActiv 
		AND GVL_PrintingBed.PrintingBed.bAtTemp THEN
			eState := E_StateSequencer.PREP_PRINTING_HEX_6;
		END_IF
		
	// =============================================================================
	E_StateSequencer.PREP_PRINTING_HEX_6 : // Buffer leeren
	// =============================================================================
		IF FC_Execute('CLEAR_PROG_BUFFER','') THEN 
			IF bAbort THEN
				eState := E_StateSequencer.ABORTED;
			ELSE
				eState := E_StateSequencer.PREP_PRINTING_HEX_7;
			END_IF
		END_IF
		
	// =============================================================================
	E_StateSequencer.PREP_PRINTING_HEX_7 : // Druckprozess gestartet (Hexapod auf Startposition fahren)
	// =============================================================================
		IF FC_Execute('GEO_LINE','LA 0 0 -305 0 0 0') THEN // Position 0 0 -105
			IF bAbort THEN
				eState := E_StateSequencer.ABORTED;
			ELSE
				eState := E_StateSequencer.READ_FILE;
			END_IF
		END_IF
	
	// =============================================================================
	E_StateSequencer.READ_FILE : // Zeile aus File lesen
	// =============================================================================
		IF bStopExtOnBlockEnd AND FC_WaitForFinish() THEN
		// Extruder muss am Blockende gestoppt werden, obwohl gerade noch Zeilen für den nächsten Block eingelesen werden
			eState := E_StateSequencer.STOP_EXTRUDING;
		ELSIF NOT bPause AND NOT bAbort THEN
		// Zeile lesen, wenn nicht Pause oder Abbruch
			// Zeile lesen
			IF bFirstRunState THEN 
				fbReadFile(
					sNetId := '',
					hFile := hFile,
					bExecute := TRUE, 
					tTimeout := T#5S);
			ELSE
				fbReadFile(bExecute := FALSE);
			END_IF
			
			// Fehler
			IF fbReadFile.bError THEN
			bError := TRUE;
			nErrorID := 3003;
			sErrorMsg := 'Datei: Fehler beim lesen der aktuellen Zeile';
			END_IF
			
			// Ergebnis auslesen im 2. Cycle
			IF NOT bFirstRunState AND NOT fbReadFile.bBusy AND NOT fbReadFile.bError THEN
				IF NOT fbReadFile.bEOF THEN
				// Nicht am Dateiende
					sLine := fbReadFile.sLine;
					eState := E_StateSequencer.EXECUTE_LINE;
				ELSE
				// Dateiende erreicht
					sLine := '';
					eState := E_StateSequencer.FINISHED;
				END_IF
			END_IF
		ELSIF bAbort THEN
			eState := E_StateSequencer.ABORTED;
		ELSIF bPause THEN
			eState := E_StateSequencer.PAUSE;
		END_IF
	
	// =============================================================================
	E_StateSequencer.EXECUTE_LINE : // Zeile ausführen
	// =============================================================================
		sLineTrimmed := FC_Trim(sLine);
		// Unterscheidung Verfahrweg und Extrusion
		IF sLineTrimmed = 'EXTRUDER_OFF' THEN
			IF bBlockWithExt THEN 
				eState := E_StateSequencer.EXTRUDER_OFF_1;
			ELSE
				// Zeile: EXTRUDER_OFF, obwohl Extruder bereits aus ist
				eState := E_StateSequencer.READ_FILE;
			END_IF
		ELSIF sLineTrimmed = 'EXTRUDER_ON' THEN
			IF NOT bBlockWithExt THEN 
				eState := E_StateSequencer.EXTRUDER_ON_1;
			ELSE
				// Zeile: EXTRUDER_ON, obwohl Extruder bereits an ist
				eState := E_StateSequencer.READ_FILE;
			END_IF
		ELSIF sLineTrimmed = '' THEN
			eState := E_StateSequencer.READ_FILE;
		ELSIF bProgBlockStart THEN
			// Erste Zeile im Programmblock
			eState := E_StateSequencer.WRITE_KOS;
		ELSE
			eState := E_StateSequencer.WRITE_PROG;
		END_IF
	
	// =============================================================================
	E_StateSequencer.WRITE_KOS : // Koordinatensystem in Programm an Hexabridge schreiben (wird zu Programmstart zurückgesetzt)
	// =============================================================================	
		// Erste Programmzeile: Koordinatensystem schreiben
		IF bAbort THEN
			eState := E_StateSequencer.ABORTED;
		ELSE
			IF FC_WriteProgLine('SK Extruder')THEN
				eState := E_StateSequencer.WRITE_FEED;
			END_IF
		END_IF
	
	// =============================================================================
	E_StateSequencer.WRITE_FEED : // Vorschub in Programm an Hexabridge schreiben
	// =============================================================================	
		// Zweite Programmzeile: Vorschub schreiben (Extrudieren oder Verfahren)
		IF bAbort THEN
			eState := E_StateSequencer.ABORTED;
		ELSIF bBlockWithExt THEN
			IF FC_WriteProgLine(CONCAT('VF ',TO_STRING(fFeed * 60))) THEN
				bProgBlockStart := FALSE;
				eState := E_StateSequencer.WRITE_PROG;
			END_IF
		ELSE
			IF FC_WriteProgLine(CONCAT('VF ',TO_STRING(fTravelFeed * 60)))THEN
				bProgBlockStart := FALSE;
				eState := E_StateSequencer.WRITE_PROG;
			END_IF
		END_IF
		
	// =============================================================================
	E_StateSequencer.WRITE_PROG : // Bewegnungszeile in Programm an Hexabridge schreiben
	// =============================================================================	
		// Programmzeile hinzufügen
		IF bAbort THEN
			eState := E_StateSequencer.ABORTED;
		ELSIF FC_WriteProgLine(sLineTrimmed) THEN
			eState := E_StateSequencer.READ_FILE;
		END_IF
	
	
	// =============================================================================
	E_StateSequencer.EXTRUDER_ON_1 : // Extruder abschalten nach vorherigen Block
	// =============================================================================
		// Laufender Prgrammblock ist mit Extruder an (2 Segmente vor der aktuellen Zeile)
		// Warte bis dieser fertig ist und schalte Extruder ab
		// Starte dann den bis hier eingelsenen Block im Eilgang (Extruder aus)
		IF bAbort THEN
			eState := E_StateSequencer.ABORTED;
		ELSIF FC_WaitForFinish() THEN
			IF bStopExtOnBlockEnd THEN
				bBackToExtruderOn2 := TRUE;
				eState := E_StateSequencer.STOP_EXTRUDING;
			ELSE
				eState := E_StateSequencer.EXTRUDER_ON_2;
			END_IF
		END_IF
		

	// =============================================================================
	E_StateSequencer.EXTRUDER_ON_2 : // Progammblock ausführen 	
	// =============================================================================
		// Bis jetzt geschriebener Progammblock ist also mit Extruder OFF
		GVL_Hexabridge.bProgLineExecution := TRUE;
		
		IF FC_ExecuteNoWait('RUN_PROG_BUFFER','') THEN
			// Extruder in nächsten Block an
			bBlockWithExt := TRUE;
			bProgBlockStart := TRUE;
			eState := E_StateSequencer.READ_FILE;
		END_IF
		
		
	// =============================================================================	
	E_StateSequencer.EXTRUDER_OFF_1 : // Warte bis vorheriger Block beendet
	// =============================================================================
		// Bis jetzt geschriebener Progammblock ist also mit Extruder ON --> Anschalten
		IF bAbort THEN
			eState := E_StateSequencer.ABORTED;
		ELSIF FC_WaitForFinish() THEN
			eState := E_StateSequencer.START_EXTRUDING;
		END_IF
		
	// =============================================================================	
	E_StateSequencer.START_EXTRUDING : // Extrusion starten
	// =============================================================================
		GVL_Extruder.Extruder.bStop := FALSE;
		GVL_Extruder.Extruder.bStart := TRUE;
		bPrintBedClear := FALSE;
		
		IF bAbort THEN
			eState := E_StateSequencer.ABORTED;
		ELSIF GVL_Extruder.Extruder.bExtruding THEN
			bStopExtOnBlockEnd := TRUE;
			eState := E_StateSequencer.EXTRUDER_OFF_2;
		END_IF
	
	// =============================================================================	
	E_StateSequencer.EXTRUDER_OFF_2 : // Progammblock ausführen
	// =============================================================================
		// Bis jetzt geschriebenen Progammblock ausführen
		GVL_Hexabridge.bProgLineExecution := TRUE;
		
		IF FC_ExecuteNoWait('RUN_PROG_BUFFER','') THEN
			// Extruder im nächsten Block aus
			bBlockWithExt := FALSE;
			bProgBlockStart := TRUE;
			eState := E_StateSequencer.READ_FILE;
		END_IF
		
		
	// =============================================================================	
	E_StateSequencer.STOP_EXTRUDING : // Extrusion stoppen, wenn Ende des Prgrammblocks erreicht
	// =============================================================================
		GVL_Extruder.Extruder.bStop := TRUE;
		GVL_Extruder.Extruder.bStart := FALSE;
		IF NOT GVL_Extruder.Extruder.bExtruding THEN
			// Extruder gestoppt
			bStopExtOnBlockEnd := FALSE;
			IF bBackToExtruderOn2 THEN
				bBackToExtruderOn2 := FALSE;
				eState := E_StateSequencer.EXTRUDER_ON_2;
			ELSIF bBackToPause THEN
				bBackToPause := FALSE;
				eState := E_StateSequencer.PAUSE;
			ELSE
				eState := E_StateSequencer.READ_FILE;	
			END_IF
		END_IF
		

	// =============================================================================
	E_StateSequencer.PAUSE : // Druck pausiert
	// =============================================================================
		// Warte bis der Block ausgeführt wurde und schalte wenn nötig am Ende den Extruder ab
		IF bStopExtOnBlockEnd THEN
			IF FC_WaitForFinish() THEN
				bBackToPause := TRUE;
				eState := E_StateSequencer.STOP_EXTRUDING;
			END_IF
		END_IF

		IF bResume THEN			
			bPause := FALSE;
			bResume := FALSE;
			eState := E_StateSequencer.READ_FILE;
		END_IF
	
	// =============================================================================
	E_StateSequencer.ABORTED : // Druckprozess abgebrochen
	// =============================================================================
		GVL_Extruder.Extruder.bStopHeater := TRUE;
		GVL_Extruder.Extruder.bStop := TRUE;
		
		GVL_HexaBridge.bProgLineSaved := FALSE;
		GVL_HexaBridge.sProgLine := '';
		GVL_HexaBridge.bProgLineReady := FALSE;
		
		IF FC_WaitForFinish() THEN
			bAbort := FALSE;
			eState := E_StateSequencer.SHUTDOWN;
		END_IF
		
	// =============================================================================
	E_StateSequencer.FINISHED : // Ende der Datei --> Letzten Programmblock ausführen
	// =============================================================================
		// Bis jetzt geschriebener ProgammBlock ist also mit Extruder OFF
		GVL_Hexabridge.bProgLineExecution := TRUE;
		
		IF FC_Execute('RUN_PROG_BUFFER','') THEN
			bFinished := TRUE;
			eState := E_StateSequencer.SHUTDOWN;
		END_IF
			
	// =============================================================================
	E_StateSequencer.SHUTDOWN : // Herunterfahren
	// =============================================================================
		// Status
		bReady := FALSE;
	
		// Schalte Extruder ab
		GVL_Extruder.Extruder.bStopHeater := TRUE;
		GVL_PrintingBed.PrintingBed.fSetTemp := 0.0;
		
		// Hexapod einfahren
		IF NOT bError THEN
			IF FC_Execute('GEO_LINE','PU') THEN
				eState := E_StateSequencer.CLOSE_FILE;
			END_IF
		END_IF
END_CASE;

METHOD FC_Trim : STRING(255)
VAR_INPUT
	sString			: STRING(255);
END_VAR
VAR
	sWithoutLF		: STRING(255);
	sWithoutLFCR	: STRING(255);
	sLF				: STRING(5)			:= '$N';
	sCR				: STRING(5)			:= '$R';
END_VAR
// Entfernt Leerzeichen und Absätze
FindAndDelete(
	pSrcString		:= ADR(sString),
	pDeleteString	:= ADR(sLF),
	pDstString		:= ADR(sWithoutLF),
	nDstSize		:= SIZEOF(sWithoutLF));
	
// FindAndDelete(
// 	pSrcString		:= ADR(sWithoutLF),
// 	pDeleteString	:= ADR(sCR),
// 	pDstString		:= ADR(sWithoutLFCR),
// 	nDstSize		:= SIZEOF(sWithoutLFCR));
 
FC_Trim := F_LTRIM(F_RTRIM(sWithoutLF));
END_METHOD

END_FUNCTION_BLOCK

// ---- POUs/HexaBridge/FC_Execute.TcPOU
FUNCTION FC_Execute : BOOL
VAR_INPUT
	sCommand			: STRING(MAX_STRING_LENGTH);	// Befehl
	sParam				: STRING(MAX_STRING_LENGTH);	// Parameter
END_VAR
VAR
	sCommandTrimmed		: STRING(MAX_STRING_LENGTH);	// Entfernt Leerzeichen
	sParamTrimmed		: STRING(MAX_STRING_LENGTH);	// Entfernt Leerzeichen
END_VAR

IF GVL_HexaBridge.bHexConnected AND GVL_HexaBridge.bBridgeRunning THEN
	// Senden des Befehls
	IF NOT GVL_HexaBridge.bDone AND NOT GVL_HexaBridge.bBusy
	AND NOT GVL_HexaBridge.bCommandSent AND NOT GVL_HexaBridge.bExecute THEN
		// Befehl senden
		sCommandTrimmed := F_LTRIM(F_RTRIM(sCommand));
		sParamTrimmed := F_LTRIM(F_RTRIM(sParam));
		GVL_HexaBridge.sCommand := sCommandTrimmed;
		GVL_HexaBridge.sGeoLine := sParamTrimmed;
		GVL_Hexabridge.bExecute := TRUE;
		GVL_HexaBridge.bCommandSent := TRUE;
	END_IF
	
	// Empfangen des Ergebnisses der Ausführung des Befehls
	IF GVL_HexaBridge.bCommandSent AND NOT GVL_HexaBridge.bExecute
	AND GVL_HexaBridge.bDone AND NOT GVL_HexaBridge.bBusy THEN
		GVL_HexaBridge.bDone := FALSE;
		GVL_HexaBridge.bCommandSent := FALSE;
		IF NOT GVL_HexaBridge.bError THEN
			FC_Execute := TRUE;
		ELSE 
			FC_Execute := FALSE;
		END_IF
	END_IF
END_IF

END_FUNCTION

// ---- POUs/HexaBridge/FC_WaitForFinish.TcPOU
FUNCTION FC_WaitForFinish : BOOL
VAR_INPUT
END_VAR
VAR
END_VAR

IF GVL_HexaBridge.bHexConnected AND GVL_HexaBridge.bBridgeRunning THEN
	// Empfangen des Ergebnisses der Ausführung des Befehls
	IF GVL_HexaBridge.bCommandSent AND NOT GVL_HexaBridge.bExecute
	AND GVL_HexaBridge.bDone AND NOT GVL_HexaBridge.bBusy THEN
		GVL_HexaBridge.bDone := FALSE;
		GVL_HexaBridge.bCommandSent := FALSE;
		IF NOT GVL_HexaBridge.bError THEN
			FC_WaitForFinish := TRUE;
		ELSE 
			FC_WaitForFinish := FALSE;
		END_IF
	ELSIF NOT GVL_HexaBridge.bCommandSent AND NOT GVL_HexaBridge.bExecute
	AND NOT GVL_HexaBridge.bDone AND NOT GVL_HexaBridge.bBusy THEN
		FC_WaitForFinish := TRUE;
	END_IF
END_IF

END_FUNCTION

// ---- POUs/HexaBridge/FC_WriteProgLine.TcPOU
FUNCTION FC_WriteProgLine : BOOL
VAR_INPUT
	sLine			: STRING(MAX_STRING_LENGTH);	// GeoCode Befehl
END_VAR
VAR
END_VAR

IF GVL_HexaBridge.bHexConnected AND GVL_HexaBridge.bBridgeRunning THEN
	// Senden des Befehls
	IF GVL_HexaBridge.sProgLine = '' AND NOT GVL_HexaBridge.bProgLineReady AND GVL_HexaBridge.bProgLineSaved
	AND NOT GVL_HexaBridge.bExecute AND NOT GVL_HexaBridge.bProgLineExecution THEN
		GVL_HexaBridge.bProgLineSaved := FALSE;
		GVL_HexaBridge.sProgLine := sLine;
		GVL_HexaBridge.bProgLineReady := TRUE;
		FC_WriteProgLine := TRUE;
	END_IF
END_IF

END_FUNCTION

// ---- POUs/HexaBridge/FC_ExecuteNoWait.TcPOU
FUNCTION FC_ExecuteNoWait : BOOL
VAR_INPUT
	sCommand			: STRING(MAX_STRING_LENGTH);	// Befehl
	sParam				: STRING(MAX_STRING_LENGTH);	// Parameter
END_VAR
VAR
	sCommandTrimmed		: STRING(MAX_STRING_LENGTH);	// Entfernt Leerzeichen
	sParamTrimmed		: STRING(MAX_STRING_LENGTH);	// Entfernt Leerzeichen
END_VAR

IF GVL_HexaBridge.bHexConnected AND GVL_HexaBridge.bBridgeRunning THEN
	// Vorheriger Befehl ausgeführt?
	IF GVL_HexaBridge.bCommandSent AND NOT GVL_HexaBridge.bExecute
	AND GVL_HexaBridge.bDone AND NOT GVL_HexaBridge.bBusy THEN
		GVL_HexaBridge.bDone := FALSE;
		GVL_HexaBridge.bCommandSent := FALSE;
	END_IF

	// Senden des Befehls
	IF NOT GVL_HexaBridge.bDone AND NOT GVL_HexaBridge.bBusy
	AND NOT GVL_HexaBridge.bCommandSent AND NOT GVL_HexaBridge.bExecute THEN

		// Befehl senden
		sCommandTrimmed := F_LTRIM(F_RTRIM(sCommand));
		sParamTrimmed := F_LTRIM(F_RTRIM(sParam));
		GVL_HexaBridge.sCommand := sCommandTrimmed;
		GVL_HexaBridge.sGeoLine := sParamTrimmed;
		GVL_Hexabridge.bExecute := TRUE;
		GVL_HexaBridge.bCommandSent := TRUE;
		
		// Ausgang
		IF NOT GVL_HexaBridge.bError THEN
			FC_ExecuteNoWait := TRUE;
		ELSE 
			FC_ExecuteNoWait := FALSE;
		END_IF
	END_IF
END_IF

END_FUNCTION

// ---- POUs/PrintingBed/FB_PrintingBedSync.TcPOU
FUNCTION_BLOCK FB_PrintingBedSync
VAR_INPUT
	bErrorReset		: BOOL;
END_VAR
VAR_OUTPUT
	// Statusinformationen
	bError        	: BOOL;				// Fehler
    nErrorID      	: UDINT;
    sErrorMsg 		: STRING(80);
END_VAR
VAR
	// ADS-Kommunikation
    fbReadADS_AtTemp	: FB_ReadAdsSymByName;
	fbReadADS_ActTemp	: FB_ReadAdsSymByName;
	fbWriteADS_SetTemp	: FB_WriteAdsSymByName;

    // Konfiguration
    sRemoteNetID		: T_AmsNetId 	:= '172.16.6.70.1.1'; 	// Ziel-AMS-NetID
    sRemotePort 		: T_AmsPort		:= 856; 				// Hexapod PLC
	tTimeout			: TIME			:= T#5S;				// Zeit bis zu ADS Timeout
	
	// Temp
	nADSErrorID			: UDINT;
	bReadBusy_AtTemp	: BOOL;
	bReadBusy_ActTemp	: BOOL;
	bWriteBusy_SetTemp	: BOOL;
	bError_AtTemp		: BOOL;
	bError_ActTemp		: BOOL;
	bError_SetTemp		: BOOL;
END_VAR

IF NOT bError OR bErrorReset THEN
fbReadADS_AtTemp(
	bRead			:= NOT bReadBusy_AtTemp,
	sNetId			:= sRemoteNetID,
	nPort			:= sRemotePort,
	sVarName		:= 'GVL_PrintingBed.Druckbett_T_valid',
	nLen			:= SIZEOF(GVL_PrintingBed.PrintingBed.bAtTemp),
	nDestAddr		:= ADR(GVL_PrintingBed.PrintingBed.bAtTemp),
	tTimeout		:= tTimeout,
	eComMode		:= E_AdsComMode.eAdsComModeFastCom,
	bClearOnError	:= bErrorReset,
	bBusy			=> bReadBusy_AtTemp,
	bError			=> bError_AtTemp,
	nErrorId		=> nADSErrorID);

fbReadADS_ActTemp(
	bRead			:= NOT bReadBusy_ActTemp,
	sNetId			:= sRemoteNetID,
	nPort			:= sRemotePort,
	sVarName		:= 'GVL_PrintingBed.Druckbett_Tist',
	nLen			:= SIZEOF(GVL_PrintingBed.PrintingBed.fActualTemp),
	nDestAddr		:= ADR(GVL_PrintingBed.PrintingBed.fActualTemp),
	tTimeout		:= tTimeout,
	eComMode		:= E_AdsComMode.eAdsComModeFastCom,
	bClearOnError	:= bErrorReset,
	bBusy			=> bReadBusy_ActTemp,
	bError			=> bError_ActTemp,
	nErrorId		=> nADSErrorID);

fbWriteADS_SetTemp(
	bWrite			:= NOT bWriteBusy_SetTemp,
	sNetId			:= sRemoteNetID,
	nPort			:= sRemotePort,
	sVarName		:= 'GVL_PrintingBed.Druckbett_Tsoll',
	nLen			:= SIZEOF(GVL_PrintingBed.PrintingBed.fSetTemp),
	nSrcAddr		:= ADR(GVL_PrintingBed.PrintingBed.fSetTemp),
	tTimeout		:= tTimeout,
	eComMode		:= E_AdsComMode.eAdsComModeFastCom,
	bBusy			=> bWriteBusy_SetTemp,
	bError			=> bError_SetTemp,
	nErrorId		=> nADSErrorID);
END_IF

bError := bError_AtTemp OR bError_ActTemp OR bError_SetTemp;

IF bErrorReset AND NOT bError THEN
	bErrorReset := FALSE;
	nErrorID := 0;
	sErrorMsg := '';
END_IF

IF bError THEN
	nErrorID := 4000;
	sErrorMsg := CONCAT('ADS Fehler: ', TO_STRING(nADSErrorID));
END_IF

END_FUNCTION_BLOCK

// ---- POUs/Extruder/FB_ExtruderControl.TcPOU
FUNCTION_BLOCK FB_ExtruderControl
VAR_INPUT
	bHeatersEnabled	: BOOL;						// Heizelemente aktiviert
END_VAR
VAR_OUTPUT
	// Statusinformationen
	bReady 			: BOOL;						// Betriebsbereit auf Temperatur
	bExtruding 		: BOOL;						// Motor läuft
	bHeatingActiv 	: BOOL;						// Heizelemente
	bError        	: BOOL;						// Fehler
    nErrorID      	: UDINT;
    sErrorMsg 		: STRING(80);
END_VAR
VAR
	// Zustandsmaschine
	eState			: E_StateExtruder := E_StateExtruder.OFF;	//State
END_VAR
VAR_IN_OUT
	// Steuersignale
	bStartHeater 	: BOOL;						// Heizelemente aktivieren
	bStopHeater		: BOOL;						// Abschalten und Abkühlen
	bStart 			: BOOL;						// Start-Befehl Extrusion
	bStop 			: BOOL;						// Stop-Befehl Extrusion
	bErrorReset 	: BOOL;						// Reset-Befehl für Fehler
END_VAR

(*
	0   - Ausgeschaltet (OFF)
	10  - Initialisierung (INIT)
	100 - Warte auf Befehl (IDLE)
	200 - Aufheizen (HEATING)
	300 - Betriebsbereit (READY)
	310 - Motor aktiviert / Drucken (PRINTING)
	400 - Herunterfahren (SHUTDOWN)
*)

// =============================================================================
// Extrusionsrate berechnen
// =============================================================================
FC_ExtrusionCalculations();

// =============================================================================
// Funktionsabhängigkeiten (Heizen vor Extrusion und Stop dominant)
// =============================================================================
IF bStop THEN
	bStart := FALSE;
ELSIF bStart THEN
	bStartHeater := TRUE;
END_IF

IF bStopHeater OR NOT bHeatersEnabled THEN
	bStart := FALSE;
	bStop := TRUE;
	bStartHeater := FALSE;
END_IF

// =============================================================================
// Fehlerbahandlung
// =============================================================================
IF bErrorReset AND bError THEN
	GVL_Extruder.HeaterTop.bErrorReset := TRUE;
	GVL_Extruder.HeaterMiddle.bErrorReset := TRUE;
	GVL_Extruder.HeaterNozzle.bErrorReset := TRUE;
	GVL_Extruder.ExtruderMotor.bErrorReset := TRUE;
	bErrorReset := FALSE;
	bError := FALSE;
END_IF;

bError := bError
	OR GVL_Extruder.HeaterTop.bError 
	OR GVL_Extruder.HeaterMiddle.bError
	OR GVL_Extruder.HeaterNozzle.bError
	OR GVL_Extruder.ExtruderMotor.bError;
	
IF bError THEN
	IF GVL_Extruder.HeaterTop.bError 		THEN nErrorID := GVL_Extruder.HeaterTop.nErrorID + 10; END_IF
	IF GVL_Extruder.HeaterMiddle.bError 	THEN nErrorID := GVL_Extruder.HeaterMiddle.nErrorID + 20; END_IF
	IF GVL_Extruder.HeaterNozzle.bError 	THEN nErrorID := GVL_Extruder.HeaterNozzle.nErrorID + 30; END_IF
	IF GVL_Extruder.ExtruderMotor.bError 	THEN nErrorID := GVL_Extruder.ExtruderMotor.nErrorID; END_IF
	IF GVL_Extruder.HeaterTop.bError 		THEN sErrorMsg := GVL_Extruder.HeaterTop.sErrorMsg; END_IF
	IF GVL_Extruder.HeaterMiddle.bError 	THEN sErrorMsg := GVL_Extruder.HeaterMiddle.sErrorMsg; END_IF
	IF GVL_Extruder.HeaterNozzle.bError 	THEN sErrorMsg := GVL_Extruder.HeaterNozzle.sErrorMsg; END_IF
	IF GVL_Extruder.ExtruderMotor.bError 	THEN sErrorMsg := GVL_Extruder.ExtruderMotor.sErrorMsg; END_IF
END_IF

IF bError AND NOT (eState = E_StateExtruder.IDLE OR eState = E_StateExtruder.OFF) THEN
	eState := E_StateExtruder.SHUTDOWN;
END_IF

// =============================================================================
// Status
// =============================================================================
bExtruding := GVL_Extruder.ExtruderMotor.bRunning;

// =============================================================================
// Zustandsmaschine
// =============================================================================
CASE eState OF
	// =============================================================================
	E_StateExtruder.OFF : // Ausgeschaltet
	// =============================================================================
		// Alles aus
		GVL_Extruder.HeaterTop.bEnabled := FALSE;
		GVL_Extruder.HeaterMiddle.bEnabled := FALSE;
		GVL_Extruder.HeaterNozzle.bEnabled := FALSE;
		GVL_Extruder.ExtruderMotor.bEnable := FALSE;
	
		// Status
		bReady := FALSE;
		bHeatingActiv := FALSE;
		
		IF NOT bError THEN
			eState := E_StateExtruder.INIT;
		END_IF;
		
	// =============================================================================
	E_StateExtruder.INIT: // Initialisierung
	// =============================================================================
		eState := E_StateExtruder.IDLE;
	
	// =============================================================================
	E_StateExtruder.IDLE : // Idle
	// =============================================================================
		// Alles aus
		GVL_Extruder.HeaterTop.bEnabled := FALSE;
		GVL_Extruder.HeaterMiddle.bEnabled := FALSE;
		GVL_Extruder.HeaterNozzle.bEnabled := FALSE;
		GVL_Extruder.ExtruderMotor.bEnable := FALSE;
	
		// Status
		bReady := FALSE;
		bHeatingActiv := FALSE;
		
		IF bStartHeater 
		AND (GVL_ParameterExtruder.aMaterialSettings[GVL_ParameterExtruder.nMaterial].fTempTop 		<> 0.0 
			OR GVL_ParameterExtruder.aMaterialSettings[GVL_ParameterExtruder.nMaterial].fTempMiddle <> 0.0 
			OR GVL_ParameterExtruder.aMaterialSettings[GVL_ParameterExtruder.nMaterial].fTempNozzle <> 0.0) 
		AND NOT bStopHeater AND bHeatersEnabled THEN
			eState := E_StateExtruder.HEATING;
		END_IF;
		
	// =============================================================================
	E_StateExtruder.HEATING : // Aufheizen
	// =============================================================================
		// Starte Heizelemente
		GVL_Extruder.HeaterTop.bEnabled := TRUE;
		GVL_Extruder.HeaterMiddle.bEnabled := TRUE;
		GVL_Extruder.HeaterNozzle.bEnabled := TRUE;
		GVL_Extruder.ExtruderMotor.bEnable := FALSE;
		
		//Status
		bReady := FALSE;
		bHeatingActiv := TRUE;
		
		// Prüfe, ob alle Temperaturen erreicht
		IF bStopHeater OR NOT bHeatersEnabled THEN
			eState := E_StateExtruder.SHUTDOWN;
		ELSIF (GVL_Extruder.HeaterTop.bAtTemp OR GVL_ParameterExtruder.aMaterialSettings[GVL_ParameterExtruder.nMaterial].fTempTop = 0.0)
		AND (GVL_Extruder.HeaterMiddle.bAtTemp OR GVL_ParameterExtruder.aMaterialSettings[GVL_ParameterExtruder.nMaterial].fTempMiddle = 0.0)
		AND (GVL_Extruder.HeaterNozzle.bAtTemp OR GVL_ParameterExtruder.aMaterialSettings[GVL_ParameterExtruder.nMaterial].fTempNozzle = 0.0) THEN
			eState := E_StateExtruder.READY;
		END_IF
	
	// =============================================================================
	E_StateExtruder.READY: // Betriebsbereit, Heizelemente aktiv
	// =============================================================================
		//Status
		bReady := TRUE;
		bHeatingActiv := TRUE;
		
		// Heizelemente aktiv
		GVL_Extruder.HeaterTop.bEnabled := TRUE;
		GVL_Extruder.HeaterMiddle.bEnabled := TRUE;
		GVL_Extruder.HeaterNozzle.bEnabled := TRUE;
		GVL_Extruder.ExtruderMotor.bEnable := FALSE;

		IF bStopHeater OR NOT bHeatersEnabled THEN
			eState := E_StateExtruder.SHUTDOWN;
		ELSIF bStart THEN
			eState := E_StateExtruder.PRINTING;
		END_IF;
	
	// =============================================================================
	E_StateExtruder.PRINTING : // Motor aktiviert / Extrusion
	// =============================================================================
		// Halte Heizungen aktiv
		GVL_Extruder.HeaterTop.bEnabled := TRUE;
		GVL_Extruder.HeaterMiddle.bEnabled := TRUE;
		GVL_Extruder.HeaterNozzle.bEnabled := TRUE;
		
		// Motor starten
		GVL_Extruder.ExtruderMotor.bEnable := TRUE;
		
		//Status
		bReady := TRUE;
		bHeatingActiv := TRUE;
		
		IF bStopHeater OR NOT bHeatersEnabled THEN
			eState := E_StateExtruder.SHUTDOWN;		
		ELSIF bStop THEN
			GVL_Extruder.ExtruderMotor.bEnable := FALSE;
			eState := E_StateExtruder.READY;
		END_IF;
	
	// =============================================================================
	E_StateExtruder.SHUTDOWN : // Herunterfahren
	// =============================================================================
		// Schalte alles ab
		GVL_Extruder.HeaterTop.bEnabled := FALSE;
		GVL_Extruder.HeaterMiddle.bEnabled := FALSE;
		GVL_Extruder.HeaterNozzle.bEnabled := FALSE;

		GVL_Extruder.ExtruderMotor.bEnable := FALSE;
		
		// Status
		bReady := FALSE;
		bHeatingActiv := FALSE;
		
		// Cooldown Bedingung (alles unter 35°C)
		IF GVL_Extruder.HeaterTop.fActualTemp < 35
		AND GVL_Extruder.HeaterMiddle.fActualTemp < 35
		AND GVL_Extruder.HeaterNozzle.fActualTemp < 35 THEN
			eState := E_StateExtruder.IDLE;
		ELSIF (GVL_ParameterExtruder.aMaterialSettings[GVL_ParameterExtruder.nMaterial].fTempTop 	<> 0.0 
		OR GVL_ParameterExtruder.aMaterialSettings[GVL_ParameterExtruder.nMaterial].fTempMiddle <> 0.0 
		OR GVL_ParameterExtruder.aMaterialSettings[GVL_ParameterExtruder.nMaterial].fTempNozzle <> 0.0) 
		AND NOT bError AND bStartHeater AND NOT bStopHeater AND bHeatersEnabled THEN
			eState := E_StateExtruder.HEATING;
		END_IF;
END_CASE;

END_FUNCTION_BLOCK

// ---- POUs/Extruder/FC_ExtrusionCalculations.TcPOU
FUNCTION FC_ExtrusionCalculations : BOOL
VAR_INPUT
END_VAR
VAR
	fCalcMaxFlow		: LREAL;
	fCalcMaxSpeed		: LREAL;
	fCalcFlowRate		: LREAL;
	fCalcMotorRPM		: LREAL;
END_VAR

// =============================================================================
// Eingaben begrenzen
// =============================================================================
GVL_ParameterExtruder.fSpeedOverride	:= LIMIT(0, GVL_ParameterExtruder.fSpeedOverride, 100);
GVL_ParameterExtruder.fSafetyMargin		:= LIMIT(0, GVL_ParameterExtruder.fSafetyMargin, 100);

// =============================================================================
// Formeln nach https://dyzedesign.com/2024/05/flow-to-rpm-factor-optimize-your-3d-printing-with-pellet-extruders/	
// =============================================================================
fCalcMaxFlow	:= 	GVL_ParameterExtruder.aMaterialSettings[GVL_ParameterExtruder.nMaterial].fMaxFlowRate 
					+ TO_LREAL(GVL_ParameterExtruder.nNozzleSize);

fCalcMaxSpeed	:= 	fCalcMaxFlow
					* LIMIT(0, GVL_ParameterExtruder.fSafetyMargin, 100) / 100
					* LIMIT(0, GVL_ParameterExtruder.fSpeedOverride, 100) / 100
					/ (GVL_ParameterExtruder.fLayerHeight
					* (GVL_ParameterExtruder.fLayerWidth - 0.215 * GVL_ParameterExtruder.fLayerHeight));
					
										
fCalcFlowRate 	:=	GVL_ParameterExtruder.fLayerHeight
					* (GVL_ParameterExtruder.fLayerWidth - 0.215 * GVL_ParameterExtruder.fLayerHeight)
					* fCalcMaxSpeed;

fCalcMotorRPM	:=	LIMIT (0, GVL_ParameterExtruder.aMaterialSettings[GVL_ParameterExtruder.nMaterial].fFlow2RPM
					* GVL_ParameterExtruder.aMaterialSettings[GVL_ParameterExtruder.nMaterial].fNozzleSizeCoef
					* fCalcFlowRate, PAR_Extruder.C_MAX_RPM_SCREW_FULL * PAR_Extruder.C_GEAR_RATIO);

// =============================================================================
// Rückrechnung wenn maximale RPM des Extruders erreicht (Schraube max. 50 RPM)
// =============================================================================
IF GVL_ParameterExtruder.fMotorRPM = PAR_Extruder.C_MAX_RPM_SCREW_FULL * PAR_Extruder.C_GEAR_RATIO THEN
	fCalcFlowRate 	:= 	PAR_Extruder.C_MAX_RPM_SCREW_FULL * PAR_Extruder.C_GEAR_RATIO 
						/ GVL_ParameterExtruder.aMaterialSettings[GVL_ParameterExtruder.nMaterial].fFlow2RPM
						/ GVL_ParameterExtruder.aMaterialSettings[GVL_ParameterExtruder.nMaterial].fNozzleSizeCoef;
										
	fCalcMaxSpeed	:= 	GVL_ParameterExtruder.fFlowRate	
						/ GVL_ParameterExtruder.fLayerHeight
						/ (GVL_ParameterExtruder.fLayerWidth - 0.215 * GVL_ParameterExtruder.fLayerHeight);					
END_IF

// =============================================================================
// Werte schreiben
// =============================================================================
GVL_ParameterExtruder.fMaximumFlow 		:= fCalcMaxFlow;
GVL_ParameterExtruder.fMaximumSpeed 	:= fCalcMaxSpeed;
GVL_ParameterExtruder.fFlowRate 		:= fCalcFlowRate;
GVL_ParameterExtruder.fMotorRPM			:= fCalcMotorRPM;

END_FUNCTION

// ---- POUs/Extruder/FB_HeaterZone.TcPOU
FUNCTION_BLOCK INTERNAL FB_HeaterZone
VAR_INPUT
	nTempRaw		: INT		:= 0;		// Rohwert (muss durch 10 geteilt werden)
	fAtTempTolerance: LREAL		:= 2;		// Toleranz für bAtTemp [K]
	
	// PID-Abtastfaktor (Vielfaches der Task-Zykluszeit)
    nPIDCycleFactor: UINT  		:= 10;		// PID rechnet alle n Zyklen

    // PID-Tuning
    fWarmupKp       : LREAL;   				// Proportionalverstärkung
    fWarmupKi       : LREAL;  				// Integralverstärkung
    fWarmupKd       : LREAL;  				// Differentialversträrkung

    // Filterfaktor für DT1-Anteil des PID-Reglers
    fWarmupFilterN  : LREAL 	:= 10.0;  	// zwischen 5 und 20 --> mehr Rauschen = kleiner
	
	tRampTime		: TIME;					// Einschaltrampendauer beim aktivieren
	
	bPrinting		:BOOL;					// Schaltete PID-Parameter um
	
	// PID-Tuning
    fPrintingKp     : LREAL;   				// Proportionalverstärkung
    fPrintingKi     : LREAL;  				// Integralverstärkung
    fPrintingKd     : LREAL;  				// Differentialversträrkung

    // Filterfaktor für DT1-Anteil des PID-Reglers
    fPrintingFilterN: LREAL 	:= 10.0;  	// zwischen 5 und 20 --> mehr Rauschen = kleiner

    // PWM-Konfiguration
    tPWM_Period   	: TIME  	:= T#5S;  	// Lange Periode, wenig Schalten, da träges System
END_VAR
VAR_OUTPUT
	fActualTemp   	: LREAL;             	// Isttemperatur [°C]
	fPID_Output    	: LREAL;				// PID-Wert
    bSSR_Out      	: BOOL;					// SSR Ein oder Aus
    bAtTemp        	: BOOL;					// Temperatur erreicht
    bError        	: BOOL;					// Fehler
    nErrorID      	: UDINT;
    sErrorMsg 		: STRING(80);
END_VAR
VAR_IN_OUT
	bEnable         : BOOL;
	bErrorReset		: BOOL;					// Fehler zurücksetzen
	fSetTemp       	: LREAL;             	// Solltemperatur [°C]
END_VAR
VAR
	// PID
	fbPID               : FB_CTRL_PID;
	stPID_Params		: ST_CTRL_PID_PARAMS;
	eMode_PID           : E_CTRL_MODE;
    
	// Einschaltrampe
	fbRampTimer				: TON;		// Timer für die Rampe
	fStartingTemp			: LREAL;	// Starttmperatur
	fRampIncrease			: LREAL;	// Anstieg der Rampe
	fbFirstCycleEnable		: R_TRIG;	// Erster Durchgang nach Einschalten
	
	// PWM
	fbPWM               : FB_CTRL_PWM_OUT;
    stPWM_Params        : ST_CTRL_PWM_OUT_PARAMS;
	eMode_PWM           : E_CTRL_MODE;
	eState_PWM			: E_CTRL_STATE;
	
	// Berechnete PID-Parameter
	tTn                 : TIME;
    tTv                 : TIME;
    tTd                 : TIME;
	fKp					: LREAL;
	
	fSetpoint			: LREAL;
	
	// Timing
    tPIDCycleTime	: TIME 	:= T#100MS;	// PID-Abtastzeit [s]
    tTaskCycleTime	: TIME  := T#10MS;	// Task-Zykluszeit
	nTaskIdx     	: DINT;
    nCycleTime   	: UDINT;
	
    // Fehlerflags
    bSensorError        : BOOL;
    bOverTempError      : BOOL;
END_VAR

// =============================================================================
// Zykluszeiten bestimmen und für FBs umrechnen
// =============================================================================
nTaskIdx := GETCURTASKINDEXEX();
IF nTaskIdx > 0 AND _TaskInfo[nTaskIdx].FirstCycle 
THEN
	nCycleTime := _TaskInfo[nTaskIdx].CycleTime;
	
	// Task-Zykluszeit für PWM
	tTaskCycleTime := UDINT_TO_TIME(nCycleTime / 10000);
	
	// PID-Abtastzeit = Task-Zykluszeit × Faktor
	tPIDCycleTime := tTaskCycleTime * nPIDCycleFactor;
END_IF

// =============================================================================
// Kp, Ki, Kd → Tn, Tv, Td umrechnen
// =============================================================================
IF bPrinting THEN
	IF fPrintingKi > 0.0 THEN
		tTn := T#0S + LREAL_TO_TIME(fPrintingKp / fPrintingKi * 1000.0);
	ELSE
		tTn := T#0S;
	END_IF
	
	IF fPrintingKp > 0.0 THEN
		tTv := T#0S + LREAL_TO_TIME(fPrintingKd / fPrintingKp * 1000.0);
	ELSE
		tTv := T#0S;
	END_IF
	
	IF fPrintingFilterN > 0.0 THEN
		tTd := T#0S +  LREAL_TO_TIME( TIME_TO_LREAL(tTv) / fPrintingFilterN);
	ELSE
		tTd := T#0S + LREAL_TO_TIME( TIME_TO_LREAL(tTv) / 10.0);
	END_IF
	
	fKp := fPrintingKp;
ELSE
	IF fWarmupKi > 0.0 THEN
		tTn := T#0S + LREAL_TO_TIME(fWarmupKp / fWarmupKi * 1000.0);
	ELSE
		tTn := T#0S;
	END_IF
	
	IF fWarmupKp > 0.0 THEN
		tTv := T#0S + LREAL_TO_TIME(fWarmupKd / fWarmupKp * 1000.0);
	ELSE
		tTv := T#0S;
	END_IF
	
	IF fWarmupFilterN > 0.0 THEN
		tTd := T#0S +  LREAL_TO_TIME( TIME_TO_LREAL(tTv) / fWarmupFilterN);
	ELSE
		tTd := T#0S + LREAL_TO_TIME( TIME_TO_LREAL(tTv) / 10.0);
	END_IF
	
	fKp := fWarmupKp;
END_IF

// =============================================================================
// Temperatur umrechnen
// =============================================================================
fActualTemp := TO_REAL(nTempRaw)/10;

// =============================================================================
// Sensorcheck
// =============================================================================
bSensorError   := (fActualTemp < PAR_Extruder.C_MIN_SENSOR_TEMP) OR (fActualTemp > PAR_Extruder.C_MAX_SENSOR_TEMP);
bOverTempError := (fActualTemp > PAR_Extruder.C_MAX_TEMP) AND NOT bSensorError;

IF bSensorError THEN
    bError    := TRUE;
    nErrorID  := 1001;
    sErrorMsg := 'Sensorfehler: Wert ausserhalb Bereich';
ELSIF bOverTempError THEN
    bError    := TRUE;
    nErrorID  := 1002;
    sErrorMsg := 'Uebertemperatur! Heizung abgeschaltet';
END_IF

// =============================================================================
// Solltemperatur begrenzen
// =============================================================================
fSetTemp := LIMIT(PAR_Extruder.C_MIN_SET_TEMP, fSetTemp, PAR_Extruder.C_MAX_SET_TEMP);

// =============================================================================
// PID-Regler (FB_BasicPID)
// =============================================================================
IF bErrorReset OR NOT bEnable THEN
	eMode_PID := eCTRL_MODE_RESET;
ELSIF bEnable AND NOT bError THEN
    eMode_PID := eCTRL_MODE_ACTIVE;
ELSE
    eMode_PID := eCTRL_MODE_PASSIVE;
END_IF

stPID_Params.tCtrlCycleTime := tPIDCycleTime;
stPID_Params.tTaskCycleTime := tTaskCycleTime;
stPID_Params.fKp := fKp;
stPID_Params.tTn := tTn;
stPID_Params.tTv := tTv;
stPID_Params.tTd := tTd;
stPID_Params.fOutMaxLimit := 100;
stPID_Params.fOutMinLimit := 0;
stPID_Params.bPInTheFeedbackPath := FALSE;
stPID_Params.bDinTheFeedbackPath := FALSE;
stPID_Params.bARWOnIPartOnly := FALSE;

// Rampe um direkte Sprünge zu verhindern und Regler zu stabilisieren
fbRampTimer(IN := bEnable, PT := tRampTime);
fbFirstCycleEnable(CLK := bEnable);
IF fbFirstCycleEnable.Q THEN
	fStartingTemp := fActualTemp;
	fRampIncrease := (fSetTemp - fStartingTemp)/ TIME_TO_LREAL(tRampTime);
END_IF

IF bEnable THEN
	IF fbRampTimer.Q THEN
		fSetpoint := fSetTemp;
	ELSE
		fSetpoint := TIME_TO_LREAL(fbRampTimer.ET) * fRampIncrease + fStartingTemp;
	END_IF
END_IF


fbPID(
    fSetpointValue  := fSetpoint,
    fActualValue    := fActualTemp,
	fManSyncValue	:= 0,
	bSync			:= FALSE,
	eMode			:= eMode_PID,
	bHold			:= FALSE,
	stParams		:= stPID_Params);
	
fPID_Output := fbPID.fOut;

IF fbPID.bError THEN
	bError    := TRUE;
	nErrorID  := 1003;
	sErrorMsg := CONCAT('PID-Regler: ', TO_STRING(fbPID.eErrorId));
END_IF

// =============================================================================
// PWM-Ausgang (FB_CTRL_PWM_OUT)
// =============================================================================
IF bErrorReset THEN
	eMode_PWM := eCTRL_MODE_RESET;
ELSIF bEnable AND NOT bError THEN
    eMode_PWM := eCTRL_MODE_ACTIVE;
ELSE
    eMode_PWM := eCTRL_MODE_PASSIVE;
END_IF

stPWM_Params.tPWMPeriod := tPWM_Period;
stPWM_Params.tTaskCycleTime := tTaskCycleTime;
stPWM_Params.bInstantPWMUpdate := TRUE;

fbPWM(
    fPWMInput	:= fPID_Output, // 3
    eMode    	:= eMode_PWM,
    stParams 	:= stPWM_Params
);
bSSR_Out := fbPWM.bPwmOutBitPos;
eState_PWM := fbPWM.eState;

IF fbPWM.bError THEN
	bError := TRUE;
	nErrorID  := 1005;
    sErrorMsg :=CONCAT('PWM: ',TO_STRING(fbPWM.eErrorId));
END_IF

// =============================================================================
// Temperatur erreicht und Fehlerbehandlung
// =============================================================================
bAtTemp := bEnable
         AND NOT bError
           AND (fSetTemp = 0.0 OR (fActualTemp >= fSetTemp - 1 AND fActualTemp <= fSetTemp + fAtTempTolerance));

IF bError THEN
    bSSR_Out    := FALSE;
    bEnable		:= FALSE;
    bAtTemp     := FALSE;
END_IF

// =============================================================================
// Fehler zurücksetzen
// =============================================================================
IF bErrorReset THEN
    bError          := FALSE;
    nErrorID        := 0;
    sErrorMsg       := '';
    bErrorReset 	:= FALSE;
END_IF

END_FUNCTION_BLOCK

// ---- POUs/Extruder/FB_MotorControl.TcPOU
FUNCTION_BLOCK INTERNAL FB_MotorControl
VAR_INPUT
    fSetRPM      		: LREAL		:= 0;       // Soll-Drehzahl [RPM]
	bError_Stepper		: BOOL;					// Fehler der Klemme EL2521
	bStepper_STALL		: BOOL;					// Stallguard aktive (Motor überlastet)
END_VAR
VAR_OUTPUT
	// Status
    bRunning       		: BOOL;					// Motor läuft
	bError        		: BOOL;					// Fehler
    nErrorID      		: UDINT;
    sErrorMsg 			: STRING(80);
	
	// Prozessdaten
	n_Direction			: INT		:= 16383;	// Entspricht 5 V --> Vorgegebene Drehrichtung
	n_Enable			: INT		:= 0;		// Entspricht 0 V --> Aktiv
	nPTO_FreqValue  	: INT		:= 0;		// PTO Control → Frequency value (Vorzeichen entspricht Richtung)
END_VAR
VAR
    fRPM				: LREAL;				// Motoro RPM
	fDisplay_RPM		: LREAL;				// HMI RPM Value
	Powering_Off		: F_TRIG;				// Fallende Flanke --> True
	bFirstCycle			: BOOL		:= TRUE;	// Erster Durchlauf
	fMaxMotorRPM		: LREAL;				// Maximale RPM
	fRatio          	: LREAL;				// Verhältnis SollRPM zu maximaler RPM [%]
END_VAR
VAR_IN_OUT
	bEnable         	: BOOL;  				// Freigabe des Motors
	bErrorReset			: BOOL;					// Fehler zurücksetzen
END_VAR

// =============================================================================
// RPM Änderung nur im ausgeschaltetem Zustand
// =============================================================================
Powering_Off(CLK := bEnable);

IF Powering_Off.Q OR bFirstCycle THEN
	fRPM := fSetRPM;
END_IF

// =============================================================================
// Stallguard aktive (Motor überlastet) --> Abschalten
// =============================================================================
IF bStepper_STALL THEN
	bError 			:= TRUE;
	nErrorID        := 2001;
    sErrorMsg       := 'Stallguard aktive (Motor überlastet)';
END_IF

// =============================================================================
// Fehler der Klemme EL2521
// =============================================================================
IF bError_Stepper THEN
	bError 			:= TRUE;
	nErrorID        := 2004;
    sErrorMsg       := 'Motoransteuerungsfehler: Klemme EL2521';
END_IF

// =============================================================================
// FB_MotorControl – EL2521 Relativer Modus
// =============================================================================
fMaxMotorRPM := PAR_Extruder.C_MAX_RPM_SCREW * PAR_Extruder.C_GEAR_RATIO;

// Fehlererkennung
IF fSetRPM < 0 THEN
	bError 			:= TRUE;
	nErrorID        := 2002;
    sErrorMsg       := 'RPM darf nicht negativ sein';
ELSIF fSetRPM > fMaxMotorRPM THEN
	bError 			:= TRUE;
	nErrorID        := 2003;
    sErrorMsg       := 'RPM überschreitet Maximalwert';
END_IF

// Verhältnis RPM zu maximaler RPM und Grenzwertbeschränkung
fRatio := LIMIT(0, fRPM, fMaxMotorRPM) / fMaxMotorRPM;

// Setzen der Drehgeschwindigkeit
IF bEnable AND fRPM > 0.01 AND NOT bError THEN
	// Motor aktivieren
	n_Enable := 0;	
	fDisplay_RPM := fRPM;
	// Relativ: 32767 = 100% Grundfrequenz
	nPTO_FreqValue := LREAL_TO_INT(fRatio * 32767.0);
    bRunning       := TRUE;
ELSE
	// Motor deaktivieren
	n_Enable := 16383;	
    nPTO_FreqValue := 0;
	fDisplay_RPM := 0;
    bRunning       := FALSE;
END_IF

// =============================================================================
//Drehrichtung festlegen (Retraction ist verboten)
// =============================================================================

IF NOT PAR_Extruder.C_STEPPER_DIR THEN
	n_Direction := 16383;
ELSE
	n_Direction := 0;
END_IF

// =============================================================================
//Fehler zurücksetzen
// =============================================================================
IF bErrorReset THEN
    bError          := FALSE;
    nErrorID        := 0;
    sErrorMsg       := '';
    bErrorReset 	:= FALSE;
END_IF

IF bFirstCycle THEN
	bFirstCycle := FALSE;
END_IF

END_FUNCTION_BLOCK

// ---- GlobalTextList.TcGTLO
TEXTLIST GlobalTextList
  892 = '%.0f'
  505 = '%.0f RPM'
  487 = '%.1f'
  322 = '%.1f RPM'
  186 = '%.1f °C'
  777 = '%.2f'
  451 = '%2.f'
  735 = '%f'
  466 = '%n'
  339 = '%s'
  815 = '%sGVL_ProgrammSequencer.Sequencer.sErrorMsg'
  650 = 'Abbrechen'
  403 = 'Datei geladen'
  962 = 'Datei laden'
  83 = 'Datei schließen'
  577 = 'Dateipfad:'
  389 = 'Druckbett Temp.'
  726 = 'Druckparameter anpassen'
  669 = 'Druckprozess abbrechen'
  266 = 'Druckprozess abgeschlossen'
  786 = 'Druckprozess fortsetzen'
  898 = 'Druckprozess kann gestartet werden'
  452 = 'Druckprozess kann gestartet werden.'
  422 = 'Druckprozess läuft'
  792 = 'Druckprozess läuft!'
  88 = 'Druckprozess pausieren'
  569 = 'Druckprozess startbereit'
  40 = 'Druckprozess starten'
  183 = 'Erfolgreich abgeschlossen'
  658 = 'Extrusion stoppen'
  500 = 'Fehler zurücksetzen'
  891 = 'Fehlerbeschreibung: %s'
  841 = 'Flow2RPM'
  319 = 'Gewähltes Material'
  150 = 'Gewähltes Material:'
  273 = 'Heizelemente aktivieren!'
  63 = 'Heizelemente freigeben'
  9 = 'Ist das Druckbett frei?'
  184 = 'Material wechseln '
  509 = 'Materialeinstellungen'
  74 = 'Max. FlowRate'
  504 = 'Name'
  1 = 'NozzleSizeCoef'
  368 = 'Override der Extrusionsrate und Vorschubs'
  853 = 'Override der Extrusionsrate und Vorschubs:'
  136 = 'Schichtbreite'
  495 = 'Schichtbreite in mm:'
  350 = 'Schichtbreite:'
  992 = 'Schichthöhe in mm: '
  939 = 'Schichthöhe: '
  693 = 'Temp. Düse'
  728 = 'Temp. Middle'
  586 = 'Temp. Mitte'
  916 = 'Temp. oben'
  110 = 'Temp. Oben'
  808 = 'Temp. Top'
  75 = 'Verfahrgeschwindigkeit in mm/s:'
  408 = 'Verfahrgeschwindigkeit:'
  385 = 'Vorbereitung'
  668 = 'zurück'
END_TEXTLIST

// ---- VISUs/V_Konfiguration.TcVIS
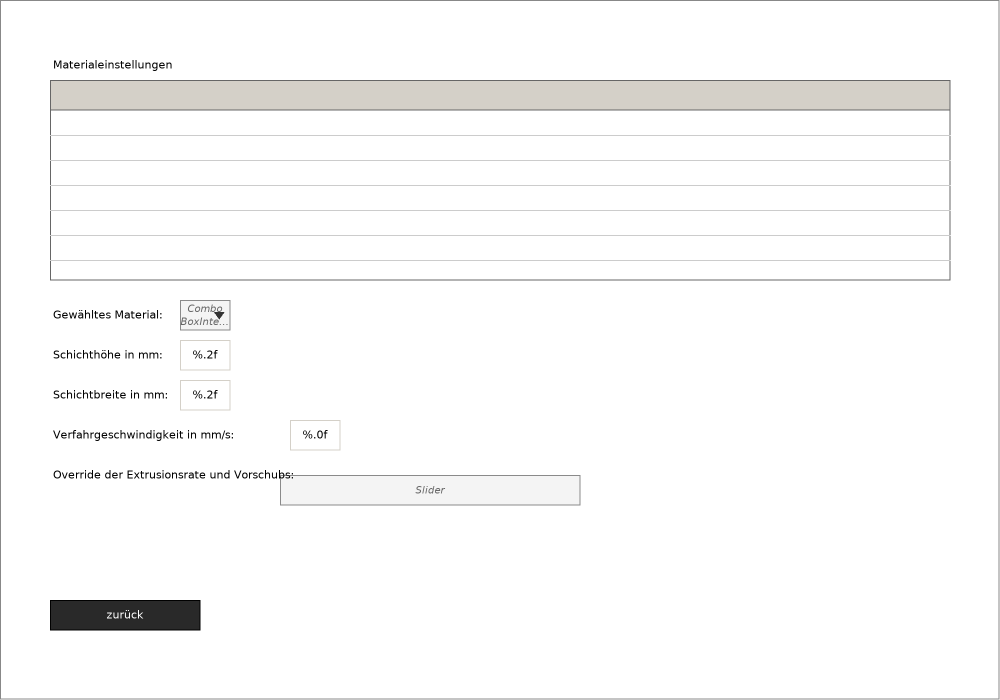
VISUALIZATION V_Konfiguration  // 1000x700
    Table (50,80 900x200), data array: GVL_ParameterExtruder.aMaterialSettings
        p3854506369: GVL_ParameterExtruder.aMaterialSettings[INDEX].sMaterial
        p1892666644: GVL_ParameterExtruder.aMaterialSettings[INDEX].fTempPrintingBed
        p338671338: GVL_ParameterExtruder.aMaterialSettings[INDEX].fTempTop
        p2170511999: GVL_ParameterExtruder.aMaterialSettings[INDEX].fTempMiddle
        p746581629: GVL_ParameterExtruder.aMaterialSettings[INDEX].fFlow2RPM
        p3104783080: GVL_ParameterExtruder.aMaterialSettings[INDEX].fNozzleSizeCoef
        p2232123230: Name
        p511219082: Druckbett Temp.
        p1755163831: Temp. Oben
        p4092479075: Temp. Mitte
        p3723444502: GVL_ParameterExtruder.aMaterialSettings[INDEX].fTempNozzle
        p2237128397: Temp. Düse
        p1218418051: GVL_ParameterExtruder.aMaterialSettings[INDEX].fMaxFlowRate
        p505689113: Max. FlowRate
    Slider (280,475 300x30), variable: GVL_ParameterExtruder.fSpeedOverride, scale 0..100
    ComboBoxInteger (180,300 50x30), variable: GVL_ParameterExtruder.nMaterial
    Label (50,50 150x30), "Materialeinstellungen"
    Label (50,300 150x30), "Gewähltes Material:"
    Label (50,340 150x30), "Schichthöhe in mm:"
    Label (50,380 150x30), "Schichtbreite in mm:"
    Label (50,460 300x30), "Override der Extrusionsrate und Vorschubs:"
    Label (50,420 200x30), "Verfahrgeschwindigkeit in mm/s:"
    Textfield (180,340 50x30), "%.2f", text variable: GVL_ParameterExtruder.fLayerHeight
    Textfield (180,380 50x30), "%.2f", text variable: GVL_ParameterExtruder.fLayerWidth
    Textfield (290,420 50x30), "%.0f", text variable: GVL_ParameterExtruder.fTravelSpeed
    Rectangle (50,600 150x30), "zurück"
        OnMouseDown: change screen: V_Homescreen
END_VISUALIZATION

// ---- VISUs/V_Homescreen.TcVIS
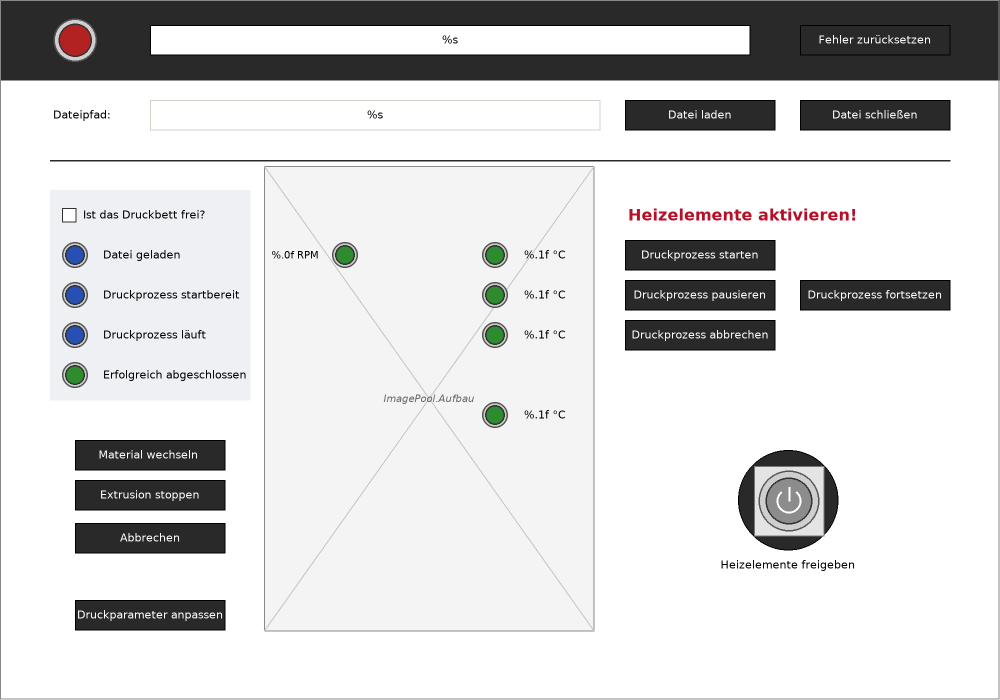
VISUALIZATION V_Homescreen  // 1000x700
    Rectangle (625,100 150x30), "Datei laden", colour toggle: GVL_ProgramSequencer.Sequencer.bLoadFile, input disabled if: Sequencer.bFileLoaded
        OnMouseDown: toggle GVL_ProgramSequencer.Sequencer.bLoadFile
    Textfield (150,100 450x30), "%s", text variable: GVL_ProgramSequencer.Sequencer.sPath
        OnMouseDown: write the text variable via Default, format %s
    Label (50,100 100x30), "Dateipfad:"
    Rectangle (800,100 150x30), "Datei schließen", colour toggle: GVL_ProgramSequencer.Sequencer.bCloseFile, input disabled if: NOT Sequencer.bFileLoaded OR GVL_ProgramSequencer.Sequencer.bPrinting
        OnMouseDown: toggle GVL_ProgramSequencer.Sequencer.bCloseFile
    Group (713,450 150x130)
        Ellipse (25,0 100x100), colour toggle: GVL_ProgramSequencer.Sequencer.bHeatersEnabled
        PowerSwitch (41,16 70x70), variable: GVL_ProgramSequencer.Sequencer.bHeatersEnabled, behaviour: TOGGLE, style: Switch-PowerSwitch-Gray
        Label (0,100 150x30), "Heizelemente freigeben"
    Rectangle (625,240 150x30), "Druckprozess starten", colour toggle: GVL_ProgramSequencer.Sequencer.bStart, invisible if: Sequencer.eState < E_StateSequencer.READY OR Sequencer.eState >= E_StateSequencer.SHUTDOWN, input disabled if: Sequencer.eState > E_StateSequencer.READY
        OnMouseDown: toggle GVL_ProgramSequencer.Sequencer.bStart
    Label (625,200 262x30), "Heizelemente aktivieren!", invisible if: GVL_ProgramSequencer.Sequencer.bHeatersEnabled OR (Sequencer.eState < E_StateSequencer.IDLE OR Sequencer.eState >= E_StateSequencer.SHUTDOWN)
    Rectangle (625,280 150x30), "Druckprozess pausieren", colour toggle: GVL_ProgramSequencer.Sequencer.bPause, invisible if: Sequencer.eState < E_StateSequencer.READY OR Sequencer.eState >= E_StateSequencer.SHUTDOWN, input disabled if: Sequencer.eState = E_StateSequencer.PAUSE
        OnMouseDown: toggle GVL_ProgramSequencer.Sequencer.bPause
    Rectangle (800,280 150x30), "Druckprozess fortsetzen", colour toggle: GVL_ProgramSequencer.Sequencer.bResume, invisible if: Sequencer.eState < E_StateSequencer.READY OR Sequencer.eState >= E_StateSequencer.SHUTDOWN, input disabled if: Sequencer.eState <> E_StateSequencer.PAUSE
        OnMouseDown: toggle GVL_ProgramSequencer.Sequencer.bResume
    Rectangle (625,320 150x30), "Druckprozess abbrechen", invisible if: Sequencer.eState < E_StateSequencer.READY OR Sequencer.eState >= E_StateSequencer.SHUTDOWN, input disabled if: GVL_ProgramSequencer.Sequencer.bAbort
        OnMouseDown: toggle GVL_ProgramSequencer.Sequencer.bAbort
    Group (0,0 1000x80)
        Rectangle (0,0 1000x80)
        Rectangle (800,25 150x30), "Fehler zurücksetzen", colour toggle: GVL_ProgramSequencer.Sequencer.bError
            OnMouseDown: execute { GVL_ProgramSequencer.Sequencer.bErrorReset := TRUE; }
        Lamp1 (50,15 50x50), variable: GVL_ProgramSequencer.Sequencer.bError, style: Lamp-Lamp1-Red
        Rectangle (150,25 600x30), "%s", text variable: GVL_ProgramSequencer.Sequencer.sErrorMsg
    Rectangle (50,160 900x1)
    Rectangle (75,600 150x30), "Druckparameter anpassen"
        OnMouseDown: change screen: V_Konfiguration
    Rectangle (75,440 150x30), "Material wechseln", colour toggle: GVL_ProgramSequencer.Sequencer.bResume, invisible if: Sequencer.eState >= E_StateSequencer.READY, input disabled if: Sequencer.eState <> E_StateSequencer.IDLE
        OnMouseDown: toggle GVL_ProgramSequencer.Sequencer.bChangeMaterial
    Rectangle (50,190 200x210)
    Label (100,280 140x30), "Druckprozess startbereit"
    Lamp1 (60,280 30x30), variable: GVL_ProgramSequencer.Sequencer.bPrintBedClear AND GVL_ProgramSequencer.Sequencer.bReady, style: Lamp-Lamp1-Blue
    Label (100,320 140x30), "Druckprozess läuft"
    Lamp1 (60,320 30x30), variable: GVL_ProgramSequencer.Sequencer.bPrinting, style: Lamp-Lamp1-Blue
    Label (100,360 140x30), "Erfolgreich abgeschlossen"
    Lamp1 (60,360 30x30), variable: GVL_ProgramSequencer.Sequencer.bFinished, style: Lamp-Lamp1-Green
    Label (100,240 140x30), "Datei geladen"
    Lamp1 (60,240 30x30), variable: Sequencer.bFileLoaded, style: Lamp-Lamp1-Blue
    Checkbox (60,200 185x30), "Ist das Druckbett frei?", variable: GVL_ProgramSequencer.Sequencer.bPrintBedClear
    Rectangle (75,480 150x30), "Extrusion stoppen", colour toggle: GVL_ProgramSequencer.Sequencer.bResume, invisible if: Sequencer.eState >= E_StateSequencer.READY, input disabled if: Sequencer.eState <> E_StateSequencer.CHANGE_MATERIAL_2
        OnMouseDown: toggle GVL_ProgramSequencer.Sequencer.bChangeMaterialFinished
    Image (264,166 330x465), image: ImagePool.Aufbau
    Lamp1 (330,240 30x30), variable: GVL_Extruder.Extruder.bExtruding, style: Lamp-Lamp1-Green
    Rectangle (75,523 150x30), "Abbrechen", invisible if: Sequencer.eState >= E_StateSequencer.READY, input disabled if: Sequencer.eState <= E_StateSequencer.IDLE
        OnMouseDown: toggle GVL_ProgramSequencer.Sequencer.bAbort
    Rectangle (520,240 50x30), "%.1f °C", text variable: GVL_Extruder.HeaterTop.fActualTemp
    Rectangle (520,280 50x30), "%.1f °C", text variable: GVL_Extruder.HeaterMiddle.fActualTemp
    Rectangle (520,320 50x30), "%.1f °C", text variable: GVL_Extruder.HeaterNozzle.fActualTemp
    Lamp1 (480,240 30x30), variable: GVL_Extruder.HeaterTop.bAtTemp, style: Lamp-Lamp1-Green
    Lamp1 (480,280 30x30), variable: GVL_Extruder.HeaterMiddle.bAtTemp, style: Lamp-Lamp1-Green
    Lamp1 (480,320 30x30), variable: GVL_Extruder.HeaterNozzle.bAtTemp, style: Lamp-Lamp1-Green
    Rectangle (270,240 50x30), "%.0f RPM", text variable: ExtruderMotor.fDisplay_RPM
    Rectangle (520,400 50x30), "%.1f °C", text variable: GVL_PrintingBed.PrintingBed.fActualTemp
    Lamp1 (480,400 30x30), variable: GVL_PrintingBed.PrintingBed.bAtTemp, style: Lamp-Lamp1-Green
END_VISUALIZATION
